C07272=1088.319,-113.427,-50.311,174.390,16.610,152.665
C07273=1088.312,-113.696,-50.301,174.388,16.610,152.665
C07274=1088.306,-113.946,-50.291,174.386,16.608,152.665
C07275=1088.300,-114.196,-50.282,174.384,16.608,152.666
C07276=1088.294,-114.446,-50.272,174.383,16.608,152.666
C07277=1088.288,-114.696,-50.263,174.381,16.607,152.666
C07278=1088.282,-114.945,-50.253,174.380,16.606,152.666
C07279=1088.275,-115.195,-50.244,174.378,16.605,152.666
C07280=1088.269,-115.445,-50.234,174.377,16.605,152.667
C07281=1088.263,-115.695,-50.224,174.375,16.604,152.667
C07282=1088.257,-115.945,-50.215,174.373,16.603,152.667
C07283=1088.251,-116.194,-50.205,174.372,16.603,152.667
C07284=1088.245,-116.444,-50.196,174.370,16.603,152.667
C07285=1088.239,-116.693,-50.187,174.369,16.602,152.668
C07286=1088.233,-116.943,-50.177,174.368,16.602,152.668
C07287=1088.227,-117.193,-50.167,174.366,16.601,152.668
C07288=1088.220,-117.443,-50.158,174.364,16.600,152.668
C07289=1088.215,-117.693,-50.149,174.363,16.600,152.668
C07290=1088.208,-117.943,-50.139,174.361,16.599,152.669
C07291=1088.202,-118.193,-50.130,174.359,16.598,152.669
C07292=1088.197,-118.442,-50.121,174.358,16.598,152.669
C07293=1088.190,-118.691,-50.112,174.356,16.597,152.669
C07294=1088.184,-118.941,-50.102,174.355,16.596,152.669
C07295=1088.177,-119.191,-50.093,174.354,16.596,152.670
C07296=1088.171,-119.441,-50.083,174.352,16.596,152.670
C07297=1088.165,-119.691,-50.073,174.350,16.595,152.670
C07298=1088.159,-119.941,-50.065,174.348,16.594,152.670
C07299=1088.153,-120.191,-50.055,174.347,16.594,152.670
C07300=1088.147,-120.440,-50.046,174.345,16.593,152.671
C07301=1088.141,-120.689,-50.037,174.343,16.592,152.671
C07302=1088.134,-120.939,-50.027,174.342,16.592,152.671
C07303=1088.128,-121.189,-50.018,174.340,16.592,152.671
C07304=1088.122,-121.439,-50.009,174.340,16.591,152.671
C07305=1088.116,-121.689,-49.999,174.338,16.590,152.672
C07306=1088.110,-121.939,-49.990,174.336,16.590,152.672
C07307=1088.104,-122.188,-49.981,174.335,16.590,152.672
C07308=1088.098,-122.438,-49.972,174.333,16.589,152.672
C07309=1088.091,-122.687,-49.962,174.331,16.588,152.673
C07310=1088.086,-122.938,-49.953,174.330,16.588,152.673
C07311=1088.079,-123.188,-49.944,174.328,16.587,152.673
C07312=1088.074,-123.437,-49.934,174.326,16.586,152.673
C07313=1088.068,-123.686,-49.925,174.325,16.586,152.673
C07314=1088.061,-123.937,-49.917,174.323,16.586,152.674
C07315=1088.055,-124.186,-49.907,174.322,16.585,152.674
C07316=1088.049,-124.436,-49.897,174.321,16.585,152.674
C07317=1088.042,-124.686,-49.888,174.319,16.584,152.674
C07318=1088.037,-124.936,-49.879,174.317,16.583,152.674
C07319=1088.030,-125.185,-49.870,174.316,16.583,152.675
C07320=1088.024,-125.435,-49.861,174.314,16.583,152.675
C07321=1088.018,-125.685,-49.851,174.312,16.582,152.675
C07322=1088.012,-125.935,-49.842,174.311,16.582,152.675
C07323=1088.006,-126.184,-49.834,174.309,16.581,152.676
C07324=1088.000,-126.434,-49.824,174.308,16.581,152.676
C07325=1087.993,-126.684,-49.815,174.306,16.580,152.676
C07326=1087.987,-126.934,-49.806,174.304,16.580,152.676
C07327=1087.981,-127.183,-49.797,174.303,16.580,152.677
C07328=1087.974,-127.433,-49.787,174.302,16.579,152.677
C07329=1087.969,-127.683,-49.779,174.300,16.578,152.677
C07330=1087.962,-127.941,-49.769,174.299,16.578,152.677
C07331=1087.957,-128.198,-49.760,174.297,16.577,152.677
C07332=1087.958,-128.455,-49.748,174.296,16.575,152.677
C07333=1087.965,-128.710,-49.735,174.296,16.571,152.676
C07334=1087.560,-128.731,-49.860,174.254,16.677,152.705
C07335=1087.553,-128.477,-49.873,174.254,16.681,152.706
C07336=1087.552,-128.220,-49.885,174.255,16.683,152.706
C07337=1087.558,-127.963,-49.895,174.257,16.684,152.706
C07338=1087.564,-127.705,-49.904,174.258,16.684,152.705
C07339=1087.571,-127.455,-49.914,174.260,16.685,152.705
C07340=1087.576,-127.205,-49.922,174.262,16.686,152.705
C07341=1087.582,-126.955,-49.932,174.263,16.686,152.705
C07342=1087.589,-126.706,-49.941,174.265,16.687,152.705
C07343=1087.595,-126.456,-49.950,174.267,16.687,152.704
C07344=1087.601,-126.206,-49.959,174.268,16.687,152.704
C07345=1087.607,-125.957,-49.969,174.270,16.688,152.704
C07346=1087.614,-125.707,-49.978,174.271,16.689,152.704
C07347=1087.619,-125.457,-49.986,174.272,16.689,152.703
C07348=1087.626,-125.207,-49.996,174.274,16.690,152.703
C07349=1087.632,-124.957,-50.005,174.275,16.690,152.703
C07350=1087.639,-124.708,-50.014,174.277,16.691,152.703
C07351=1087.644,-124.458,-50.023,174.279,16.691,152.703
C07352=1087.650,-124.208,-50.033,174.280,16.691,152.702
C07353=1087.656,-123.958,-50.042,174.282,16.692,152.702
C07354=1087.663,-123.709,-50.051,174.284,16.693,152.702
C07355=1087.669,-123.458,-50.060,174.285,16.693,152.702
C07356=1087.675,-123.209,-50.069,174.287,16.694,152.701
C07357=1087.681,-122.960,-50.079,174.289,16.694,152.701
C07358=1087.687,-122.710,-50.088,174.289,16.695,152.701
C07359=1087.693,-122.460,-50.098,174.291,16.696,152.701
C07360=1087.700,-122.210,-50.106,174.293,16.696,152.701
C07361=1087.706,-121.960,-50.116,174.294,16.697,152.701
C07362=1087.711,-121.711,-50.125,174.296,16.697,152.700
C07363=1087.718,-121.461,-50.134,174.298,16.698,152.700
C07364=1087.724,-121.211,-50.144,174.299,16.698,152.700
C07365=1087.730,-120.961,-50.153,174.301,16.699,152.700
C07366=1087.736,-120.711,-50.162,174.303,16.700,152.699
C07367=1087.743,-120.462,-50.171,174.304,16.700,152.699
C07368=1087.748,-120.213,-50.181,174.305,16.701,152.699
C07369=1087.754,-119.963,-50.190,174.307,16.701,152.699
C07370=1087.761,-119.713,-50.200,174.308,16.701,152.699
C07371=1087.767,-119.463,-50.209,174.310,16.702,152.698
C07372=1087.773,-119.213,-50.218,174.312,16.703,152.698
C07373=1087.779,-118.963,-50.228,174.313,16.703,152.698
C07374=1087.785,-118.713,-50.237,174.315,16.704,152.698
C07375=1087.792,-118.464,-50.246,174.316,16.705,152.698
C07376=1087.798,-118.215,-50.255,174.318,16.705,152.697
C07377=1087.804,-117.965,-50.265,174.319,16.706,152.697
C07378=1087.810,-117.715,-50.275,174.321,16.706,152.697
C07379=1087.816,-117.465,-50.284,174.323,16.708,152.697
C07380=1087.822,-117.215,-50.294,174.324,16.708,152.697
C07381=1087.828,-116.966,-50.303,174.326,16.708,152.696
C07382=1087.835,-116.716,-50.313,174.327,16.709,152.696
C07383=1087.840,-116.465,-50.322,174.329,16.709,152.696
C07384=1087.847,-116.216,-50.331,174.330,16.710,152.696
C07385=1087.852,-115.967,-50.340,174.332,16.711,152.696
C07386=1087.858,-115.717,-50.350,174.333,16.711,152.696
C07387=1087.864,-115.467,-50.360,174.335,16.712,152.695
C07388=1087.871,-115.217,-50.369,174.337,16.713,152.695
C07389=1087.877,-114.967,-50.379,174.338,16.714,152.695
C07390=1087.883,-114.718,-50.388,174.339,16.714,152.695
C07391=1087.889,-114.468,-50.398,174.341,16.714,152.695
C07392=1087.895,-114.218,-50.407,174.343,16.716,152.694
C07393=1087.902,-113.968,-50.417,174.344,16.716,152.694
C07394=1087.908,-113.718,-50.427,174.346,16.717,152.694
C07395=1087.915,-113.448,-50.437,174.348,16.717,152.694
C07396=1087.921,-113.177,-50.447,174.349,16.718,152.694
C07397=1087.928,-112.907,-50.458,174.351,16.719,152.693
C07398=1087.934,-112.635,-50.468,174.353,16.720,152.693
C07399=1087.940,-112.385,-50.477,174.354,16.720,152.693
C07400=1087.947,-112.135,-50.487,174.356,16.721,152.693
C07401=1087.953,-111.886,-50.497,174.358,16.722,152.693
C07402=1087.959,-111.636,-50.506,174.359,16.722,152.693
C07403=1087.964,-111.387,-50.515,174.360,16.723,152.692
C07404=1087.971,-111.137,-50.525,174.362,16.724,152.692
C07405=1087.977,-110.887,-50.534,174.364,16.725,152.692
C07406=1087.983,-110.638,-50.545,174.365,16.725,152.692
C07407=1087.989,-110.388,-50.554,174.367,16.726,152.692
C07408=1087.995,-110.138,-50.564,174.368,16.726,152.691
C07409=1088.001,-109.888,-50.574,174.369,16.727,152.691
C07410=1088.007,-109.639,-50.584,174.371,16.728,152.691
C07411=1088.013,-109.389,-50.593,174.373,16.729,152.691
C07412=1088.020,-109.139,-50.603,174.375,16.729,152.691
C07413=1088.026,-108.889,-50.612,174.376,16.730,152.691
C07414=1088.032,-108.639,-50.622,174.377,16.730,152.690
C07415=1088.038,-108.390,-50.631,174.379,16.731,152.690
C07416=1088.045,-108.140,-50.642,174.381,16.732,152.690
C07417=1088.051,-107.891,-50.651,174.382,16.733,152.690
C07418=1088.057,-107.641,-50.661,174.383,16.734,152.690
C07419=1088.062,-107.391,-50.671,174.385,16.734,152.690
C07420=1088.068,-107.141,-50.681,174.387,16.735,152.689
C07421=1088.075,-106.891,-50.690,174.388,16.735,152.689
C07422=1088.081,-106.642,-50.700,174.390,16.737,152.689
C07423=1088.087,-106.392,-50.710,174.392,16.737,152.689
C07424=1088.093,-106.142,-50.720,174.393,16.738,152.689
C07425=1088.099,-105.892,-50.730,174.394,16.739,152.689
C07426=1088.105,-105.642,-50.739,174.396,16.739,152.688
C07427=1088.111,-105.393,-50.749,174.398,16.740,152.688
C07428=1088.118,-105.143,-50.759,174.400,16.741,152.688
C07429=1088.123,-104.893,-50.769,174.400,16.742,152.688
C07430=1088.129,-104.643,-50.779,174.402,16.743,152.688
C07431=1088.136,-104.394,-50.788,174.404,16.743,152.688
C07432=1088.142,-104.145,-50.799,174.406,16.744,152.687
C07433=1088.147,-103.894,-50.809,174.407,16.746,152.687
C07434=1088.154,-103.645,-50.818,174.408,16.746,152.687
C07435=1088.160,-103.395,-50.828,174.410,16.747,152.687
C07436=1088.166,-103.145,-50.838,174.412,16.747,152.687
C07437=1088.172,-102.896,-50.848,174.413,16.748,152.687
C07438=1088.178,-102.646,-50.858,174.414,16.749,152.687
C07439=1088.184,-102.396,-50.868,174.416,16.750,152.686
C07440=1088.190,-102.147,-50.878,174.418,16.751,152.686
C07441=1088.196,-101.897,-50.888,174.419,16.752,152.686
C07442=1088.202,-101.647,-50.898,174.421,16.752,152.686
C07443=1088.208,-101.397,-50.907,174.422,16.753,152.686
C07444=1088.215,-101.148,-50.917,174.424,16.754,152.686
C07445=1088.220,-100.898,-50.928,174.426,16.755,152.685
C07446=1088.226,-100.648,-50.937,174.427,16.756,152.685
C07447=1088.233,-100.399,-50.947,174.428,16.756,152.685
C07448=1088.238,-100.149,-50.958,174.430,16.757,152.685
C07449=1088.244,-99.899,-50.967,174.432,16.758,152.685
C07450=1088.251,-99.650,-50.977,174.433,16.759,152.685
C07451=1088.257,-99.400,-50.987,174.435,16.760,152.684
C07452=1088.263,-99.150,-50.997,174.436,16.760,152.684
C07453=1088.269,-98.901,-51.008,174.438,16.761,152.684
C07454=1088.275,-98.651,-51.017,174.440,16.762,152.684
C07455=1088.281,-98.401,-51.027,174.441,16.763,152.684
C07456=1088.288,-98.151,-51.038,174.443,16.764,152.684
C07457=1088.294,-97.901,-51.047,174.444,16.765,152.684
C07458=1088.300,-97.652,-51.058,174.446,16.765,152.684
C07459=1088.306,-97.375,-51.069,174.447,16.766,152.683
C07460=1088.312,-97.099,-51.080,174.449,16.767,152.683
C07461=1088.319,-96.822,-51.091,174.451,16.769,152.683
C07462=1088.326,-96.546,-51.103,174.452,16.769,152.683
C07463=1088.331,-96.296,-51.113,174.454,16.770,152.683
C07464=1088.338,-96.047,-51.123,174.456,16.771,152.683
C07465=1088.343,-95.796,-51.133,174.457,16.772,152.683
C07466=1088.349,-95.547,-51.143,174.458,16.773,152.683
C07467=1088.356,-95.296,-51.154,174.460,16.774,152.682
C07468=1088.362,-95.047,-51.164,174.462,16.775,152.682
C07469=1088.368,-94.797,-51.174,174.463,16.776,152.682
C07470=1088.374,-94.547,-51.184,174.465,16.777,152.682
C07471=1088.380,-94.298,-51.194,174.467,16.778,152.682
C07472=1088.386,-94.048,-51.205,174.468,16.778,152.682
C07473=1088.392,-93.799,-51.215,174.469,16.779,152.681
C07474=1088.398,-93.549,-51.225,174.471,16.780,152.681
C07475=1088.403,-93.299,-51.235,174.473,16.781,152.681
C07476=1088.410,-93.050,-51.245,174.474,16.782,152.681
C07477=1088.415,-92.799,-51.256,174.476,16.784,152.681
C07478=1088.422,-92.550,-51.266,174.477,16.784,152.681
C07479=1088.427,-92.300,-51.276,174.479,16.785,152.681
C07480=1088.434,-92.050,-51.287,174.480,16.786,152.681
C07481=1088.440,-91.801,-51.298,174.482,16.787,152.680
C07482=1088.446,-91.551,-51.307,174.484,16.788,152.680
C07483=1088.452,-91.301,-51.318,174.485,16.789,152.680
C07484=1088.458,-91.052,-51.328,174.486,16.789,152.680
C07485=1088.464,-90.802,-51.338,174.488,16.790,152.680
C07486=1088.470,-90.552,-51.348,174.490,16.791,152.680
C07487=1088.475,-90.303,-51.359,174.491,16.792,152.680
C07488=1088.482,-90.053,-51.368,174.493,16.794,152.680
C07489=1088.488,-89.803,-51.380,174.494,16.795,152.679
C07490=1088.494,-89.553,-51.391,174.495,16.795,152.679
C07491=1088.500,-89.304,-51.400,174.497,16.796,152.679
C07492=1088.506,-89.054,-51.411,174.499,16.797,152.679
C07493=1088.512,-88.804,-51.421,174.500,16.798,152.679
C07494=1088.518,-88.555,-51.431,174.502,16.799,152.679
C07495=1088.524,-88.306,-51.442,174.504,16.800,152.679
C07496=1088.530,-88.055,-51.452,174.505,16.801,152.679
C07497=1088.537,-87.806,-51.463,174.506,16.802,152.679
C07498=1088.542,-87.556,-51.473,174.508,16.803,152.678
C07499=1088.548,-87.306,-51.484,174.509,16.804,152.678
C07500=1088.554,-87.057,-51.494,174.511,16.805,152.678
C07501=1088.560,-86.806,-51.504,174.513,16.806,152.678
C07502=1088.567,-86.557,-51.515,174.515,16.807,152.678
C07503=1088.572,-86.307,-51.526,174.516,16.808,152.678
C07504=1088.578,-86.057,-51.536,174.517,16.809,152.678
C07505=1088.584,-85.808,-51.546,174.519,16.810,152.678
C07506=1088.590,-85.559,-51.557,174.520,16.811,152.677
C07507=1088.597,-85.308,-51.567,174.522,16.812,152.677
C07508=1088.603,-85.059,-51.578,174.524,16.813,152.677
C07509=1088.608,-84.809,-51.589,174.525,16.814,152.677
C07510=1088.615,-84.560,-51.599,174.527,16.815,152.677
C07511=1088.621,-84.309,-51.609,174.529,16.816,152.677
C07512=1088.627,-84.060,-51.620,174.530,16.816,152.677
C07513=1088.633,-83.810,-51.631,174.531,16.817,152.677
C07514=1088.639,-83.560,-51.641,174.533,16.819,152.676
C07515=1088.645,-83.311,-51.651,174.534,16.820,152.676
C07516=1088.651,-83.061,-51.662,174.536,16.821,152.676
C07517=1088.657,-82.812,-51.673,174.538,16.822,152.676
C07518=1088.663,-82.562,-51.683,174.539,16.823,152.676
C07519=1088.669,-82.312,-51.694,174.541,16.824,152.676
C07520=1088.676,-82.062,-51.704,174.542,16.825,152.676
C07521=1088.682,-81.813,-51.715,174.543,16.826,152.676
C07522=1088.688,-81.563,-51.726,174.545,16.827,152.676
C07523=1088.695,-81.289,-51.737,174.547,16.828,152.676
C07524=1088.701,-81.015,-51.749,174.548,16.829,152.675
C07525=1088.707,-80.740,-51.761,174.551,16.831,152.675
C07526=1088.715,-80.466,-51.772,174.553,16.831,152.675
C07527=1088.721,-80.216,-51.783,174.553,16.832,152.675
C07528=1088.727,-79.966,-51.793,174.555,16.833,152.675
C07529=1088.733,-79.717,-51.804,174.557,16.834,152.675
C07530=1088.739,-79.467,-51.815,174.558,16.835,152.675
C07531=1088.745,-79.217,-51.826,174.560,16.836,152.675
C07532=1088.751,-78.968,-51.837,174.561,16.838,152.675
C07533=1088.756,-78.718,-51.848,174.563,16.839,152.674
C07534=1088.763,-78.468,-51.857,174.565,16.840,152.674
C07535=1088.769,-78.218,-51.869,174.566,16.841,152.674
C07536=1088.775,-77.969,-51.879,174.568,16.842,152.674
C07537=1088.780,-77.719,-51.890,174.570,16.843,152.674
C07538=1088.786,-77.470,-51.901,174.570,16.844,152.674
C07539=1088.793,-77.220,-51.912,174.572,16.845,152.674
C07540=1088.799,-76.970,-51.923,174.574,16.846,152.674
C07541=1088.805,-76.721,-51.934,174.575,16.847,152.674
C07542=1088.810,-76.471,-51.945,174.577,16.848,152.674
C07543=1088.816,-76.220,-51.955,174.578,16.850,152.673
C07544=1088.822,-75.971,-51.966,174.580,16.851,152.673
C07545=1088.828,-75.722,-51.977,174.582,16.852,152.673
C07546=1088.835,-75.472,-51.987,174.583,16.853,152.673
C07547=1088.841,-75.222,-51.998,174.585,16.854,152.673
C07548=1088.846,-74.973,-52.009,174.587,16.855,152.673
C07549=1088.852,-74.723,-52.020,174.588,16.856,152.673
C07550=1088.859,-74.473,-52.031,174.590,16.858,152.673
C07551=1088.864,-74.223,-52.042,174.591,16.859,152.673
C07552=1088.870,-73.974,-52.053,174.592,16.859,152.673
C07553=1088.876,-73.724,-52.064,174.594,16.861,152.673
C07554=1088.882,-73.474,-52.075,174.595,16.862,152.672
C07555=1088.888,-73.225,-52.086,174.597,16.863,152.672
C07556=1088.894,-72.975,-52.097,174.599,16.864,152.672
C07557=1088.900,-72.725,-52.108,174.600,16.865,152.672
C07558=1088.906,-72.476,-52.119,174.602,16.867,152.672
C07559=1088.911,-72.226,-52.130,174.603,16.868,152.672
C07560=1088.917,-71.977,-52.141,174.605,16.869,152.672
C07561=1088.923,-71.726,-52.152,174.606,16.870,152.672
C07562=1088.929,-71.477,-52.163,174.608,16.871,152.672
C07563=1088.935,-71.228,-52.174,174.609,16.873,152.672
C07564=1088.941,-70.978,-52.185,174.611,16.874,152.672
C07565=1088.947,-70.728,-52.196,174.613,16.875,152.672
C07566=1088.953,-70.478,-52.207,174.614,16.876,152.671
C07567=1088.958,-70.229,-52.218,174.616,16.877,152.671
C07568=1088.964,-69.978,-52.230,174.617,16.879,152.671
C07569=1088.970,-69.729,-52.240,174.619,16.880,152.671
C07570=1088.976,-69.479,-52.251,174.621,16.881,152.671
C07571=1088.982,-69.230,-52.263,174.622,16.882,152.671
C07572=1088.988,-68.980,-52.274,174.623,16.883,152.671
C07573=1088.994,-68.731,-52.285,174.624,16.884,152.671
C07574=1088.999,-68.481,-52.296,174.626,16.885,152.671
C07575=1089.006,-68.231,-52.307,174.628,16.886,152.671
C07576=1089.012,-67.982,-52.318,174.629,16.887,152.671
C07577=1089.017,-67.732,-52.329,174.631,16.889,152.671
C07578=1089.023,-67.482,-52.341,174.632,16.890,152.671
C07579=1089.029,-67.232,-52.352,174.634,16.891,152.671
C07580=1089.035,-66.983,-52.364,174.636,16.892,152.670
C07581=1089.041,-66.733,-52.374,174.637,16.893,152.670
C07582=1089.047,-66.484,-52.385,174.639,16.895,152.670
C07583=1089.053,-66.233,-52.397,174.640,16.896,152.670
C07584=1089.059,-65.984,-52.407,174.642,16.897,152.670
C07585=1089.065,-65.734,-52.418,174.643,16.898,152.670
C07586=1089.071,-65.485,-52.430,174.645,16.900,152.670
C07587=1089.077,-65.213,-52.443,174.646,16.901,152.670
C07588=1089.084,-64.941,-52.455,174.648,16.902,152.670
C07589=1089.090,-64.668,-52.467,174.650,16.904,152.670
C07590=1089.097,-64.396,-52.479,174.652,16.905,152.670
C07591=1089.102,-64.147,-52.490,174.654,16.906,152.669
C07592=1089.109,-63.897,-52.501,174.655,16.908,152.670
C07593=1089.114,-63.647,-52.513,174.657,16.909,152.669
C07594=1089.120,-63.398,-52.525,174.658,16.910,152.669
C07595=1089.126,-63.148,-52.536,174.660,16.911,152.669
C07596=1089.132,-62.898,-52.547,174.661,16.913,152.669
C07597=1089.138,-62.648,-52.558,174.663,16.914,152.669
C07598=1089.144,-62.399,-52.570,174.665,16.915,152.669
C07599=1089.150,-62.149,-52.581,174.666,16.916,152.669
C07600=1089.156,-61.899,-52.592,174.668,16.918,152.669
C07601=1089.162,-61.650,-52.604,174.669,16.919,152.669
C07602=1089.168,-61.400,-52.615,174.671,16.920,152.669
C07603=1089.174,-61.151,-52.626,174.672,16.921,152.669
C07604=1089.180,-60.901,-52.638,174.674,16.922,152.669
C07605=1089.185,-60.651,-52.649,174.675,16.924,152.669
C07606=1089.192,-60.401,-52.661,174.677,16.925,152.668
C07607=1089.198,-60.152,-52.672,174.679,16.926,152.668
C07608=1089.204,-59.902,-52.683,174.680,16.927,152.668
C07609=1089.210,-59.653,-52.694,174.682,16.929,152.668
C07610=1089.215,-59.403,-52.707,174.683,16.930,152.668
C07611=1089.222,-59.153,-52.718,174.685,16.931,152.668
C07612=1089.227,-58.904,-52.729,174.686,16.932,152.668
C07613=1089.234,-58.654,-52.741,174.688,16.933,152.668
C07614=1089.239,-58.404,-52.752,174.690,16.935,152.668
C07615=1089.245,-58.154,-52.763,174.691,16.936,152.668
C07616=1089.251,-57.905,-52.775,174.693,16.937,152.668
C07617=1089.258,-57.655,-52.786,174.694,16.938,152.668
C07618=1089.264,-57.406,-52.798,174.696,16.939,152.668
C07619=1089.269,-57.156,-52.810,174.697,16.941,152.668
C07620=1089.275,-56.907,-52.821,174.699,16.942,152.668
C07621=1089.282,-56.657,-52.832,174.700,16.943,152.667
C07622=1089.287,-56.407,-52.843,174.702,16.944,152.667
C07623=1089.293,-56.157,-52.856,174.704,16.946,152.667
C07624=1089.300,-55.907,-52.867,174.705,16.947,152.667
C07625=1089.306,-55.658,-52.879,174.707,16.948,152.667
C07626=1089.312,-55.408,-52.890,174.708,16.949,152.667
C07627=1089.317,-55.159,-52.902,174.710,16.951,152.667
C07628=1089.324,-54.909,-52.913,174.711,16.952,152.667
C07629=1089.330,-54.660,-52.925,174.713,16.953,152.667
C07630=1089.336,-54.410,-52.936,174.715,16.954,152.667
C07631=1089.341,-54.161,-52.948,174.716,16.956,152.667
C07632=1089.348,-53.910,-52.960,174.718,16.957,152.667
C07633=1089.354,-53.661,-52.972,174.719,16.958,152.667
C07634=1089.360,-53.411,-52.982,174.721,16.959,152.667
C07635=1089.366,-53.161,-52.995,174.722,16.961,152.667
C07636=1089.372,-52.912,-53.006,174.724,16.962,152.666
C07637=1089.378,-52.662,-53.018,174.725,16.963,152.666
C07638=1089.383,-52.412,-53.029,174.727,16.965,152.666
C07639=1089.390,-52.163,-53.041,174.728,16.966,152.666
C07640=1089.396,-51.913,-53.053,174.730,16.967,152.666
C07641=1089.402,-51.664,-53.065,174.732,16.968,152.666
C07642=1089.408,-51.414,-53.077,174.734,16.970,152.666
C07643=1089.414,-51.164,-53.088,174.735,16.971,152.666
C07644=1089.421,-50.915,-53.100,174.737,16.972,152.666
C07645=1089.426,-50.664,-53.111,174.738,16.974,152.666
C07646=1089.432,-50.416,-53.123,174.740,16.975,152.666
C07647=1089.438,-50.166,-53.135,174.742,16.976,152.666
C07648=1089.444,-49.916,-53.146,174.743,16.978,152.666
C07649=1089.450,-49.666,-53.159,174.745,16.979,152.666
C07650=1089.456,-49.417,-53.170,174.746,16.980,152.666
C07651=1089.462,-49.146,-53.184,174.748,16.982,152.666
C07652=1089.469,-48.875,-53.196,174.749,16.983,152.666
C07653=1089.474,-48.604,-53.209,174.751,16.985,152.666
C07654=1089.481,-48.334,-53.221,174.753,16.986,152.665
C07655=1089.487,-48.084,-53.234,174.754,16.988,152.665
C07656=1089.494,-47.834,-53.246,174.756,16.989,152.665
C07657=1089.499,-47.584,-53.257,174.758,16.990,152.665
C07658=1089.505,-47.335,-53.269,174.759,16.991,152.665
C07659=1089.510,-47.086,-53.282,174.761,16.992,152.665
C07660=1089.517,-46.835,-53.293,174.762,16.994,152.665
C07661=1089.522,-46.586,-53.305,174.764,16.995,152.665
C07662=1089.529,-46.337,-53.317,174.765,16.996,152.665
C07663=1089.534,-46.086,-53.329,174.768,16.998,152.665
C07664=1089.540,-45.837,-53.341,174.769,17.000,152.665
C07665=1089.546,-45.587,-53.353,174.770,17.001,152.665
C07666=1089.552,-45.338,-53.365,174.772,17.002,152.665
C07667=1089.558,-45.088,-53.376,174.774,17.003,152.665
C07668=1089.564,-44.838,-53.389,174.775,17.005,152.665
C07669=1089.569,-44.589,-53.401,174.777,17.006,152.665
C07670=1089.576,-44.339,-53.413,174.778,17.008,152.665
C07671=1089.581,-44.089,-53.425,174.780,17.009,152.665
C07672=1089.587,-43.840,-53.436,174.781,17.010,152.665
C07673=1089.593,-43.590,-53.449,174.783,17.012,152.665
C07674=1089.599,-43.341,-53.461,174.784,17.013,152.664
C07675=1089.605,-43.091,-53.473,174.786,17.014,152.665
C07676=1089.611,-42.841,-53.485,174.788,17.016,152.664
C07677=1089.617,-42.592,-53.497,174.789,17.018,152.664
C07678=1089.623,-42.342,-53.509,174.791,17.019,152.664
C07679=1089.629,-42.092,-53.522,174.793,17.020,152.664
C07680=1089.635,-41.843,-53.533,174.794,17.021,152.664
C07681=1089.640,-41.593,-53.545,174.796,17.022,152.664
C07682=1089.646,-41.343,-53.558,174.797,17.024,152.664
C07683=1089.652,-41.094,-53.569,174.799,17.025,152.664
C07684=1089.658,-40.844,-53.582,174.800,17.026,152.664
C07685=1089.665,-40.595,-53.594,174.802,17.028,152.664
C07686=1089.670,-40.345,-53.606,174.803,17.029,152.664
C07687=1089.676,-40.096,-53.619,174.806,17.031,152.664
C07688=1089.683,-39.845,-53.630,174.807,17.032,152.664
C07689=1089.688,-39.596,-53.642,174.809,17.034,152.664
C07690=1089.694,-39.346,-53.655,174.810,17.035,152.664
C07691=1089.700,-39.097,-53.666,174.812,17.036,152.664
C07692=1089.706,-38.847,-53.679,174.813,17.038,152.664
C07693=1089.712,-38.598,-53.691,174.815,17.039,152.664
C07694=1089.717,-38.348,-53.704,174.816,17.040,152.664
C07695=1089.724,-38.098,-53.716,174.818,17.042,152.664
C07696=1089.729,-37.849,-53.728,174.820,17.044,152.664
C07697=1089.735,-37.599,-53.740,174.822,17.045,152.663
C07698=1089.741,-37.349,-53.753,174.823,17.046,152.663
C07699=1089.747,-37.100,-53.765,174.825,17.048,152.663
C07700=1089.753,-36.851,-53.777,174.826,17.049,152.663
C07701=1089.759,-36.601,-53.790,174.828,17.050,152.663
C07702=1089.764,-36.351,-53.802,174.829,17.052,152.663
C07703=1089.770,-36.102,-53.814,174.831,17.053,152.663
C07704=1089.776,-35.852,-53.827,174.832,17.055,152.663
C07705=1089.781,-35.602,-53.838,174.834,17.056,152.663
C07706=1089.788,-35.352,-53.850,174.836,17.058,152.663
C07707=1089.794,-35.103,-53.864,174.837,17.059,152.663
C07708=1089.800,-34.853,-53.876,174.839,17.061,152.663
C07709=1089.805,-34.604,-53.888,174.840,17.062,152.663
C07710=1089.811,-34.354,-53.901,174.842,17.063,152.663
C07711=1089.817,-34.104,-53.914,174.843,17.064,152.663
C07712=1089.823,-33.854,-53.926,174.845,17.066,152.663
C07713=1089.829,-33.606,-53.938,174.847,17.068,152.663
C07714=1089.835,-33.356,-53.950,174.848,17.069,152.663
C07715=1089.841,-33.085,-53.964,174.850,17.070,152.663
C07716=1089.847,-32.815,-53.978,174.851,17.072,152.663
C07717=1089.854,-32.544,-53.991,174.854,17.074,152.663
C07718=1089.860,-32.273,-54.004,174.855,17.075,152.663
C07719=1089.866,-32.024,-54.017,174.857,17.076,152.663
C07720=1089.872,-31.774,-54.030,174.858,17.078,152.663
C07721=1089.878,-31.525,-54.042,174.860,17.079,152.663
C07722=1089.883,-31.275,-54.054,174.862,17.081,152.663
C07723=1089.889,-31.025,-54.067,174.864,17.082,152.663
C07724=1089.895,-30.775,-54.080,174.865,17.084,152.663
C07725=1089.901,-30.527,-54.091,174.867,17.085,152.662
C07726=1089.907,-30.277,-54.104,174.868,17.087,152.663
C07727=1089.913,-30.027,-54.117,174.870,17.088,152.662
C07728=1089.919,-29.778,-54.129,174.871,17.089,152.662
C07729=1089.925,-29.528,-54.142,174.873,17.091,152.662
C07730=1089.931,-29.278,-54.154,174.875,17.092,152.662
C07731=1089.937,-29.029,-54.167,174.876,17.094,152.662
C07732=1089.943,-28.779,-54.180,174.878,17.095,152.662
C07733=1089.949,-28.529,-54.193,174.879,17.096,152.662
C07734=1089.955,-28.280,-54.205,174.881,17.098,152.662
C07735=1089.960,-28.030,-54.218,174.882,17.099,152.662
C07736=1089.966,-27.780,-54.230,174.885,17.101,152.662
C07737=1089.972,-27.531,-54.243,174.886,17.102,152.662
C07738=1089.979,-27.282,-54.255,174.888,17.103,152.662
C07739=1089.985,-27.032,-54.268,174.889,17.105,152.662
C07740=1089.990,-26.782,-54.280,174.891,17.106,152.662
C07741=1089.996,-26.532,-54.294,174.892,17.108,152.662
C07742=1090.001,-26.283,-54.306,174.894,17.109,152.662
C07743=1090.007,-26.033,-54.319,174.896,17.111,152.662
C07744=1090.013,-25.783,-54.331,174.898,17.112,152.662
C07745=1090.019,-25.534,-54.345,174.899,17.114,152.662
C07746=1090.025,-25.284,-54.357,174.900,17.115,152.662
C07747=1090.030,-25.035,-54.369,174.902,17.116,152.662
C07748=1090.037,-24.786,-54.383,174.903,17.118,152.662
C07749=1090.043,-24.536,-54.395,174.906,17.120,152.662
C07750=1090.048,-24.286,-54.408,174.907,17.121,152.662
C07751=1090.054,-24.036,-54.421,174.909,17.122,152.662
C07752=1090.060,-23.787,-54.434,174.910,17.124,152.662
C07753=1090.065,-23.537,-54.446,174.912,17.125,152.662
C07754=1090.071,-23.287,-54.459,174.914,17.127,152.662
C07755=1090.077,-23.038,-54.472,174.915,17.129,152.662
C07756=1090.083,-22.788,-54.485,174.917,17.130,152.661
C07757=1090.089,-22.539,-54.498,174.918,17.132,152.662
C07758=1090.095,-22.289,-54.511,174.920,17.133,152.661
C07759=1090.100,-22.039,-54.524,174.921,17.134,152.661
C07760=1090.106,-21.790,-54.537,174.924,17.136,152.661
C07761=1090.112,-21.541,-54.549,174.925,17.138,152.661
C07762=1090.118,-21.291,-54.562,174.927,17.139,152.661
C07763=1090.124,-21.041,-54.575,174.928,17.140,152.661
C07764=1090.129,-20.791,-54.588,174.930,17.141,152.661
C07765=1090.136,-20.542,-54.601,174.931,17.143,152.661
C07766=1090.141,-20.292,-54.614,174.933,17.145,152.661
C07767=1090.148,-20.043,-54.627,174.935,17.146,152.661
C07768=1090.154,-19.793,-54.640,174.936,17.147,152.661
C07769=1090.158,-19.544,-54.653,174.938,17.149,152.661
C07770=1090.164,-19.294,-54.666,174.939,17.151,152.661
C07771=1090.170,-19.044,-54.678,174.942,17.152,152.661
C07772=1090.176,-18.795,-54.692,174.943,17.154,152.661
C07773=1090.182,-18.545,-54.704,174.945,17.155,152.661
C07774=1090.189,-18.296,-54.718,174.946,17.157,152.661
C07775=1090.194,-18.046,-54.731,174.948,17.158,152.661
C07776=1090.200,-17.796,-54.744,174.950,17.160,152.661
C07777=1090.206,-17.546,-54.756,174.951,17.161,152.661
C07778=1090.212,-17.297,-54.770,174.953,17.163,152.661
C07779=1090.218,-17.026,-54.784,174.954,17.164,152.661
C07780=1090.225,-16.755,-54.798,174.957,17.166,152.661
C07781=1090.231,-16.484,-54.812,174.958,17.167,152.661
C07782=1090.237,-16.213,-54.827,174.960,17.169,152.661
C07783=1090.243,-15.963,-54.840,174.962,17.170,152.661
C07784=1090.249,-15.713,-54.853,174.963,17.172,152.661
C07785=1090.255,-15.464,-54.865,174.965,17.173,152.661
C07786=1090.261,-15.214,-54.879,174.966,17.175,152.661
C07787=1090.267,-14.964,-54.892,174.968,17.176,152.661
C07788=1090.273,-14.715,-54.905,174.970,17.178,152.660
C07789=1090.278,-14.465,-54.919,174.972,17.179,152.661
C07790=1090.284,-14.215,-54.931,174.973,17.181,152.660
C07791=1090.290,-13.966,-54.945,174.975,17.182,152.660
C07792=1090.296,-13.716,-54.959,174.977,17.184,152.660
C07793=1090.302,-13.467,-54.971,174.978,17.185,152.660
C07794=1090.307,-13.217,-54.985,174.980,17.187,152.660
C07795=1090.313,-12.967,-54.998,174.981,17.188,152.660
C07796=1090.319,-12.718,-55.011,174.983,17.190,152.660
C07797=1090.325,-12.468,-55.025,174.985,17.191,152.660
C07798=1090.331,-12.218,-55.037,174.986,17.193,152.660
C07799=1090.336,-11.969,-55.051,174.988,17.194,152.660
C07800=1090.342,-11.720,-55.064,174.989,17.196,152.660
C07801=1090.348,-11.469,-55.078,174.991,17.197,152.660
C07802=1090.354,-11.220,-55.091,174.993,17.199,152.660
C07803=1090.359,-10.971,-55.105,174.995,17.201,152.660
C07804=1090.365,-10.721,-55.118,174.996,17.202,152.660
C07805=1090.371,-10.471,-55.130,174.998,17.203,152.660
C07806=1090.377,-10.222,-55.144,175.000,17.205,152.660
C07807=1090.383,-9.973,-55.158,175.001,17.207,152.660
C07808=1090.388,-9.722,-55.171,175.003,17.208,152.660
C07809=1090.394,-9.473,-55.184,175.004,17.209,152.660
C07810=1090.400,-9.224,-55.198,175.006,17.211,152.660
C07811=1090.406,-8.974,-55.211,175.008,17.212,152.660
C07812=1090.411,-8.724,-55.224,175.010,17.214,152.660
C07813=1090.418,-8.475,-55.238,175.011,17.215,152.660
C07814=1090.423,-8.225,-55.251,175.013,17.217,152.660
C07815=1090.429,-7.976,-55.265,175.015,17.218,152.660
C07816=1090.435,-7.727,-55.278,175.016,17.220,152.660
C07817=1090.441,-7.477,-55.291,175.018,17.221,152.660
C07818=1090.447,-7.227,-55.304,175.019,17.223,152.660
C07819=1090.452,-6.978,-55.318,175.022,17.224,152.660
C07820=1090.459,-6.728,-55.332,175.023,17.226,152.660
C07821=1090.464,-6.479,-55.345,175.025,17.228,152.660
C07822=1090.470,-6.230,-55.359,175.026,17.229,152.660
C07823=1090.476,-5.979,-55.372,175.028,17.230,152.660
C07824=1090.482,-5.729,-55.385,175.030,17.232,152.659
C07825=1090.488,-5.480,-55.399,175.031,17.234,152.660
C07826=1090.494,-5.231,-55.413,175.033,17.235,152.659
C07827=1090.499,-4.981,-55.426,175.034,17.236,152.660
C07828=1090.506,-4.732,-55.440,175.037,17.238,152.659
C07829=1090.511,-4.482,-55.454,175.038,17.240,152.659
C07830=1090.517,-4.233,-55.467,175.040,17.241,152.659
C07831=1090.523,-3.983,-55.481,175.041,17.242,152.659
C07832=1090.529,-3.733,-55.494,175.044,17.244,152.659
C07833=1090.535,-3.483,-55.508,175.045,17.246,152.659
C07834=1090.540,-3.234,-55.521,175.047,17.247,152.659
C07835=1090.546,-2.984,-55.535,175.048,17.248,152.659
C07836=1090.552,-2.735,-55.549,175.050,17.250,152.659
C07837=1090.557,-2.485,-55.562,175.052,17.251,152.659
C07838=1090.563,-2.236,-55.576,175.053,17.253,152.659
C07839=1090.569,-1.986,-55.590,175.055,17.254,152.659
C07840=1090.575,-1.737,-55.603,175.057,17.256,152.659
C07841=1090.580,-1.487,-55.617,175.059,17.257,152.659
C07842=1090.586,-1.238,-55.631,175.060,17.259,152.659
C07843=1090.592,-0.964,-55.646,175.062,17.261,152.659
C07844=1090.599,-0.692,-55.661,175.064,17.262,152.659
C07845=1090.605,-0.418,-55.676,175.066,17.264,152.659
C07846=1090.611,-0.146,-55.691,175.067,17.266,152.659
C07847=1090.617,0.103,-55.705,175.069,17.267,152.659
C07848=1090.623,0.353,-55.719,175.071,17.269,152.659
C07849=1090.628,0.603,-55.733,175.073,17.270,152.659
C07850=1090.635,0.852,-55.746,175.074,17.272,152.659
C07851=1090.640,1.102,-55.760,175.076,17.273,152.659
C07852=1090.645,1.351,-55.774,175.078,17.275,152.659
C07853=1090.651,1.601,-55.788,175.079,17.277,152.659
C07854=1090.656,1.851,-55.802,175.081,17.278,152.659
C07855=1090.663,2.100,-55.815,175.082,17.280,152.659
C07856=1090.669,2.350,-55.829,175.085,17.281,152.659
C07857=1090.674,2.600,-55.843,175.086,17.283,152.659
C07858=1090.680,2.849,-55.857,175.088,17.284,152.659
C07859=1090.685,3.098,-55.871,175.090,17.286,152.659
C07860=1090.692,3.347,-55.885,175.092,17.287,152.658
C07861=1090.697,3.597,-55.898,175.093,17.289,152.659
C07862=1090.703,3.847,-55.913,175.094,17.290,152.659
C07863=1090.709,4.097,-55.927,175.097,17.292,152.658
C07864=1090.714,4.346,-55.940,175.098,17.294,152.658
C07865=1090.721,4.595,-55.954,175.100,17.295,152.658
C07866=1090.726,4.845,-55.968,175.101,17.296,152.658
C07867=1090.732,5.094,-55.982,175.104,17.298,152.658
C07868=1090.738,5.345,-55.996,175.105,17.300,152.658
C07869=1090.743,5.594,-56.010,175.107,17.301,152.658
C07870=1090.749,5.844,-56.024,175.109,17.303,152.658
C07871=1090.755,6.092,-56.038,175.110,17.304,152.658
C07872=1090.761,6.343,-56.052,175.112,17.306,152.658
C07873=1090.767,6.592,-56.066,175.113,17.307,152.658
C07874=1090.772,6.842,-56.080,175.116,17.309,152.658
C07875=1090.778,7.091,-56.095,175.117,17.310,152.658
C07876=1090.783,7.340,-56.108,175.119,17.312,152.658
C07877=1090.790,7.590,-56.122,175.121,17.313,152.658
C07878=1090.796,7.840,-56.136,175.122,17.315,152.658
C07879=1090.802,8.089,-56.151,175.124,17.316,152.658
C07880=1090.807,8.338,-56.164,175.125,17.318,152.658
C07881=1090.813,8.589,-56.179,175.128,17.319,152.658
C07882=1090.819,8.838,-56.193,175.129,17.321,152.658
C07883=1090.824,9.087,-56.207,175.131,17.322,152.658
C07884=1090.830,9.337,-56.221,175.133,17.324,152.658
C07885=1090.837,9.587,-56.235,175.135,17.325,152.658
C07886=1090.842,9.836,-56.249,175.136,17.327,152.658
C07887=1090.848,10.085,-56.263,175.138,17.328,152.658
C07888=1090.854,10.335,-56.278,175.140,17.330,152.658
C07889=1090.860,10.584,-56.292,175.141,17.331,152.658
C07890=1090.865,10.834,-56.306,175.143,17.333,152.658
C07891=1090.872,11.084,-56.321,175.145,17.334,152.657
C07892=1090.877,11.333,-56.335,175.147,17.336,152.657
C07893=1090.883,11.583,-56.348,175.148,17.337,152.657
C07894=1090.889,11.833,-56.363,175.150,17.339,152.657
C07895=1090.894,12.082,-56.377,175.152,17.340,152.657
C07896=1090.901,12.331,-56.391,175.154,17.341,152.657
C07897=1090.907,12.581,-56.405,175.155,17.343,152.657
C07898=1090.913,12.831,-56.419,175.157,17.345,152.657
C07899=1090.918,13.080,-56.434,175.159,17.346,152.657
C07900=1090.924,13.330,-56.448,175.160,17.347,152.657
C07901=1090.930,13.579,-56.463,175.163,17.350,152.657
C07902=1090.936,13.828,-56.477,175.164,17.351,152.657
C07903=1090.942,14.078,-56.492,175.166,17.352,152.657
C07904=1090.947,14.328,-56.505,175.167,17.353,152.657
C07905=1090.953,14.577,-56.520,175.170,17.355,152.657
C07906=1090.959,14.827,-56.534,175.171,17.357,152.657
C07907=1090.965,15.102,-56.550,175.174,17.358,152.657
C07908=1090.972,15.376,-56.566,175.175,17.360,152.657
C07909=1090.977,15.651,-56.581,175.177,17.362,152.657
C07910=1090.985,15.926,-56.597,175.179,17.363,152.657
C07911=1090.991,16.175,-56.612,175.181,17.365,152.657
C07912=1090.995,16.425,-56.626,175.183,17.366,152.657
C07913=1091.002,16.675,-56.641,175.184,17.367,152.656
C07914=1091.007,16.924,-56.655,175.186,17.370,152.656
C07915=1091.013,17.173,-56.670,175.188,17.371,152.656
C07916=1091.019,17.423,-56.685,175.189,17.372,152.656
C07917=1091.025,17.673,-56.699,175.192,17.374,152.656
C07918=1091.031,17.922,-56.713,175.193,17.376,152.656
C07919=1091.037,18.172,-56.727,175.195,17.377,152.656
C07920=1091.042,18.421,-56.743,175.197,17.379,152.656
C07921=1091.048,18.671,-56.757,175.199,17.380,152.656
C07922=1091.054,18.920,-56.771,175.200,17.382,152.656
C07923=1091.059,19.169,-56.786,175.202,17.383,152.656
C07924=1091.065,19.420,-56.800,175.204,17.384,152.656
C07925=1091.071,19.669,-56.815,175.205,17.386,152.656
C07926=1091.076,19.918,-56.830,175.207,17.387,152.656
C07927=1091.082,20.168,-56.844,175.209,17.389,152.656
C07928=1091.088,20.417,-56.859,175.211,17.390,152.656
C07929=1091.094,20.667,-56.874,175.212,17.392,152.656
C07930=1091.100,20.916,-56.888,175.215,17.393,152.656
C07931=1091.105,21.166,-56.903,175.216,17.395,152.656
C07932=1091.111,21.415,-56.918,175.218,17.396,152.656
C07933=1091.117,21.665,-56.932,175.220,17.398,152.656
C07934=1091.123,21.914,-56.946,175.222,17.399,152.656
C07935=1091.128,22.164,-56.962,175.223,17.401,152.656
C07936=1091.134,22.413,-56.976,175.225,17.403,152.656
C07937=1091.140,22.663,-56.990,175.227,17.404,152.655
C07938=1091.145,22.912,-57.006,175.228,17.405,152.656
C07939=1091.152,23.162,-57.021,175.231,17.407,152.655
C07940=1091.157,23.411,-57.034,175.232,17.409,152.655
C07941=1091.163,23.661,-57.049,175.235,17.410,152.655
C07942=1091.168,23.910,-57.065,175.236,17.411,152.655
C07943=1091.174,24.159,-57.079,175.238,17.413,152.655
C07944=1091.180,24.410,-57.093,175.240,17.415,152.655
C07945=1091.185,24.659,-57.109,175.241,17.416,152.655
C07946=1091.192,24.909,-57.123,175.243,17.417,152.655
C07947=1091.197,25.158,-57.138,175.246,17.419,152.655
C07948=1091.203,25.407,-57.154,175.247,17.421,152.655
C07949=1091.209,25.657,-57.167,175.249,17.422,152.655
C07950=1091.215,25.907,-57.182,175.251,17.424,152.655
C07951=1091.220,26.156,-57.198,175.252,17.425,152.655
C07952=1091.226,26.406,-57.213,175.254,17.426,152.655
C07953=1091.232,26.655,-57.227,175.256,17.428,152.655
C07954=1091.238,26.905,-57.243,175.258,17.429,152.655
C07955=1091.243,27.154,-57.257,175.259,17.430,152.654
C07956=1091.250,27.404,-57.271,175.262,17.433,152.655
C07957=1091.255,27.653,-57.287,175.263,17.434,152.654
C07958=1091.261,27.903,-57.302,175.265,17.435,152.654
C07959=1091.267,28.152,-57.316,175.267,17.437,152.654
C07960=1091.273,28.402,-57.332,175.269,17.438,152.654
C07961=1091.278,28.651,-57.346,175.271,17.440,152.654
C07962=1091.284,28.901,-57.362,175.273,17.441,152.654
C07963=1091.290,29.150,-57.376,175.274,17.442,152.654
C07964=1091.295,29.399,-57.392,175.276,17.445,152.654
C07965=1091.301,29.648,-57.407,175.278,17.446,152.654
C07966=1091.306,29.898,-57.422,175.279,17.447,152.654
C07967=1091.312,30.148,-57.436,175.282,17.449,152.654
C07968=1091.317,30.397,-57.451,175.284,17.450,152.654
C07969=1091.324,30.647,-57.466,175.285,17.452,152.654
C07970=1091.329,30.896,-57.481,175.287,17.453,152.654
C07971=1091.336,31.172,-57.498,175.289,17.455,152.654
C07972=1091.342,31.449,-57.515,175.291,17.456,152.654
C07973=1091.348,31.725,-57.531,175.294,17.458,152.653
C07974=1091.354,32.002,-57.548,175.295,17.460,152.654
C07975=1091.361,32.250,-57.564,175.297,17.461,152.653
C07976=1091.366,32.500,-57.579,175.299,17.462,152.653
C07977=1091.372,32.749,-57.594,175.300,17.464,152.653
C07978=1091.378,32.999,-57.609,175.303,17.466,152.653
C07979=1091.384,33.249,-57.624,175.305,17.467,152.653
C07980=1091.389,33.498,-57.639,175.307,17.469,152.653
C07981=1091.395,33.748,-57.654,175.308,17.470,152.653
C07982=1091.401,33.997,-57.669,175.310,17.471,152.653
C07983=1091.407,34.247,-57.684,175.312,17.473,152.653
C07984=1091.412,34.496,-57.700,175.314,17.474,152.653
C07985=1091.418,34.746,-57.715,175.315,17.476,152.653
C07986=1091.424,34.996,-57.730,175.318,17.478,152.653
C07987=1091.429,35.245,-57.745,175.319,17.479,152.653
C07988=1091.436,35.494,-57.761,175.322,17.480,152.653
C07989=1091.441,35.743,-57.776,175.323,17.482,152.653
C07990=1091.447,35.993,-57.791,175.325,17.483,152.652
C07991=1091.453,36.243,-57.807,175.327,17.485,152.652
C07992=1091.458,36.492,-57.822,175.329,17.486,152.652
C07993=1091.464,36.742,-57.837,175.331,17.488,152.652
C07994=1091.470,36.990,-57.853,175.333,17.489,152.652
C07995=1091.476,37.240,-57.868,175.334,17.490,152.652
C07996=1091.482,37.490,-57.883,175.337,17.492,152.652
C07997=1091.487,37.739,-57.898,175.338,17.494,152.652
C07998=1091.493,37.989,-57.913,175.340,17.495,152.652
C07999=1091.499,38.238,-57.929,175.342,17.496,152.652
C08000=1091.504,38.487,-57.945,175.344,17.498,152.652
C08001=1091.510,38.737,-57.960,175.346,17.500,152.652
C08002=1091.515,38.986,-57.975,175.348,17.501,152.652
C08003=1091.521,39.236,-57.991,175.349,17.502,152.652
C08004=1091.527,39.486,-58.007,175.351,17.504,152.652
C08005=1091.533,39.735,-58.021,175.353,17.505,152.651
C08006=1091.538,39.985,-58.037,175.356,17.507,152.651
C08007=1091.544,40.233,-58.053,175.357,17.508,152.651
C08008=1091.549,40.483,-58.068,175.359,17.509,152.651
C08009=1091.556,40.733,-58.083,175.361,17.511,152.651
C08010=1091.561,40.982,-58.099,175.363,17.512,152.651
C08011=1091.567,41.232,-58.114,175.365,17.514,152.651
C08012=1091.572,41.482,-58.130,175.367,17.515,152.651
C08013=1091.579,41.730,-58.145,175.369,17.517,152.651
C08014=1091.584,41.980,-58.161,175.371,17.518,152.651
C08015=1091.590,42.230,-58.176,175.372,17.520,152.651
C08016=1091.595,42.478,-58.192,175.374,17.521,152.651
C08017=1091.601,42.728,-58.208,175.376,17.522,152.651
C08018=1091.607,42.978,-58.223,175.379,17.524,152.650
C08019=1091.613,43.227,-58.239,175.380,17.526,152.650
C08020=1091.618,43.477,-58.254,175.382,17.527,152.650
C08021=1091.624,43.727,-58.270,175.384,17.528,152.650
C08022=1091.629,43.975,-58.286,175.386,17.530,152.650
C08023=1091.635,44.225,-58.301,175.388,17.532,152.650
C08024=1091.641,44.475,-58.317,175.389,17.533,152.650
C08025=1091.646,44.724,-58.333,175.391,17.534,152.650
C08026=1091.653,44.973,-58.348,175.394,17.536,152.650
C08027=1091.658,45.223,-58.364,175.395,17.537,152.650
C08028=1091.663,45.472,-58.379,175.397,17.539,152.650
C08029=1091.669,45.721,-58.395,175.399,17.540,152.650
C08030=1091.675,45.971,-58.411,175.401,17.542,152.649
C08031=1091.680,46.220,-58.427,175.403,17.543,152.650
C08032=1091.686,46.470,-58.442,175.404,17.544,152.649
C08033=1091.692,46.719,-58.458,175.407,17.546,152.649
C08034=1091.697,46.969,-58.474,175.409,17.547,152.649
C08035=1091.703,47.245,-58.491,175.411,17.549,152.649
C08036=1091.710,47.522,-58.509,175.413,17.551,152.649
C08037=1091.716,47.798,-58.526,175.415,17.552,152.649
C08038=1091.722,48.075,-58.544,175.417,17.554,152.649
C08039=1091.727,48.323,-58.560,175.420,17.556,152.649
C08040=1091.733,48.573,-58.576,175.421,17.557,152.649
C08041=1091.738,48.823,-58.592,175.423,17.558,152.649
C08042=1091.744,49.072,-58.608,175.425,17.560,152.649
C08043=1091.749,49.321,-58.623,175.427,17.561,152.648
C08044=1091.755,49.571,-58.640,175.429,17.563,152.648
C08045=1091.761,49.821,-58.655,175.431,17.564,152.648
C08046=1091.767,50.070,-58.671,175.433,17.566,152.648
C08047=1091.772,50.319,-58.687,175.435,17.567,152.648
C08048=1091.778,50.569,-58.703,175.436,17.568,152.648
C08049=1091.784,50.818,-58.719,175.439,17.569,152.648
C08050=1091.790,51.067,-58.735,175.440,17.571,152.648
C08051=1091.795,51.317,-58.751,175.443,17.573,152.648
C08052=1091.801,51.566,-58.767,175.444,17.574,152.648
C08053=1091.807,51.815,-58.783,175.447,17.575,152.648
C08054=1091.812,52.065,-58.799,175.448,17.576,152.648
C08055=1091.818,52.314,-58.814,175.451,17.578,152.647
C08056=1091.824,52.563,-58.831,175.453,17.579,152.647
C08057=1091.829,52.813,-58.846,175.454,17.580,152.647
C08058=1091.835,53.063,-58.863,175.457,17.582,152.647
C08059=1091.841,53.312,-58.879,175.458,17.584,152.647
C08060=1091.846,53.562,-58.895,175.461,17.585,152.647
C08061=1091.852,53.811,-58.911,175.462,17.586,152.647
C08062=1091.858,54.060,-58.927,175.465,17.588,152.647
C08063=1091.863,54.310,-58.943,175.466,17.589,152.647
C08064=1091.869,54.560,-58.959,175.469,17.591,152.647
C08065=1091.875,54.809,-58.975,175.470,17.592,152.646
C08066=1091.881,55.058,-58.991,175.472,17.593,152.646
C08067=1091.886,55.307,-59.007,175.474,17.595,152.646
C08068=1091.892,55.556,-59.023,175.476,17.596,152.646
C08069=1091.897,55.807,-59.040,175.479,17.597,152.646
C08070=1091.903,56.056,-59.056,175.480,17.598,152.646
C08071=1091.909,56.305,-59.072,175.483,17.600,152.646
C08072=1091.915,56.555,-59.088,175.484,17.601,152.646
C08073=1091.921,56.804,-59.105,175.487,17.603,152.646
C08074=1091.927,57.054,-59.120,175.488,17.604,152.645
C08075=1091.932,57.303,-59.136,175.491,17.606,152.645
C08076=1091.938,57.552,-59.152,175.492,17.607,152.645
C08077=1091.943,57.802,-59.169,175.494,17.608,152.645
C08078=1091.949,58.051,-59.185,175.497,17.609,152.645
C08079=1091.955,58.300,-59.202,175.498,17.611,152.645
C08080=1091.961,58.550,-59.218,175.501,17.612,152.645
C08081=1091.967,58.799,-59.234,175.502,17.613,152.645
C08082=1091.973,59.048,-59.250,175.505,17.615,152.645
C08083=1091.978,59.299,-59.267,175.506,17.616,152.644
C08084=1091.984,59.548,-59.283,175.509,17.618,152.644
C08085=1091.990,59.797,-59.299,175.511,17.619,152.644
C08086=1091.996,60.047,-59.315,175.513,17.620,152.644
C08087=1092.002,60.296,-59.332,175.515,17.622,152.644
C08088=1092.007,60.545,-59.348,175.517,17.623,152.644
C08089=1092.012,60.794,-59.364,175.519,17.624,152.644
C08090=1092.018,61.044,-59.381,175.521,17.626,152.644
C08091=1092.024,61.293,-59.397,175.523,17.627,152.644
C08092=1092.030,61.542,-59.413,175.524,17.628,152.643
C08093=1092.036,61.792,-59.429,175.527,17.630,152.643
C08094=1092.041,62.041,-59.446,175.529,17.630,152.643
C08095=1092.047,62.291,-59.463,175.531,17.632,152.643
C08096=1092.053,62.540,-59.479,175.533,17.633,152.643
C08097=1092.059,62.789,-59.495,175.535,17.635,152.643
C08098=1092.064,63.039,-59.512,175.537,17.636,152.643
C08099=1092.071,63.315,-59.530,175.540,17.638,152.642
C08100=1092.078,63.591,-59.548,175.542,17.639,152.642
C08101=1092.084,63.867,-59.567,175.544,17.641,152.642
C08102=1092.091,64.144,-59.585,175.546,17.641,152.642
C08103=1092.096,64.393,-59.601,175.549,17.643,152.642
C08104=1092.103,64.642,-59.618,175.550,17.644,152.642
C08105=1092.108,64.892,-59.635,175.553,17.646,152.642
C08106=1092.114,65.141,-59.651,175.555,17.647,152.642
C08107=1092.120,65.390,-59.668,175.557,17.649,152.641
C08108=1092.125,65.640,-59.684,175.559,17.650,152.641
C08109=1092.130,65.889,-59.700,175.561,17.651,152.641
C08110=1092.136,66.138,-59.717,175.563,17.652,152.641
C08111=1092.142,66.388,-59.733,175.565,17.654,152.641
C08112=1092.148,66.637,-59.750,175.567,17.655,152.641
C08113=1092.154,66.887,-59.768,175.570,17.656,152.641
C08114=1092.160,67.136,-59.784,175.571,17.657,152.640
C08115=1092.165,67.386,-59.801,175.574,17.659,152.640
C08116=1092.171,67.635,-59.817,175.575,17.660,152.640
C08117=1092.176,67.884,-59.835,175.578,17.662,152.640
C08118=1092.182,68.134,-59.851,175.579,17.663,152.640
C08119=1092.187,68.383,-59.868,175.582,17.664,152.640
C08120=1092.193,68.633,-59.884,175.584,17.665,152.640
C08121=1092.199,68.882,-59.901,175.586,17.667,152.639
C08122=1092.205,69.131,-59.918,175.588,17.668,152.639
C08123=1092.210,69.381,-59.935,175.590,17.670,152.639
C08124=1092.216,69.630,-59.951,175.592,17.671,152.639
C08125=1092.222,69.879,-59.968,175.595,17.672,152.639
C08126=1092.228,70.128,-59.985,175.596,17.673,152.639
C08127=1092.233,70.378,-60.002,175.599,17.675,152.639
C08128=1092.239,70.627,-60.018,175.600,17.676,152.639
C08129=1092.244,70.876,-60.035,175.603,17.677,152.638
C08130=1092.250,71.126,-60.052,175.605,17.679,152.638
C08131=1092.255,71.375,-60.068,175.607,17.680,152.638
C08132=1092.261,71.625,-60.086,175.609,17.681,152.638
C08133=1092.267,71.874,-60.102,175.611,17.682,152.638
C08134=1092.272,72.124,-60.119,175.613,17.684,152.638
C08135=1092.278,72.372,-60.136,175.616,17.685,152.638
C08136=1092.284,72.623,-60.153,175.617,17.686,152.637
C08137=1092.290,72.872,-60.171,175.620,17.687,152.637
C08138=1092.296,73.121,-60.187,175.622,17.689,152.637
C08139=1092.301,73.371,-60.204,175.624,17.690,152.637
C08140=1092.306,73.620,-60.222,175.626,17.691,152.637
C08141=1092.312,73.869,-60.238,175.628,17.692,152.637
C08142=1092.318,74.118,-60.255,175.630,17.694,152.637
C08143=1092.324,74.367,-60.272,175.632,17.695,152.636
C08144=1092.329,74.617,-60.288,175.634,17.696,152.636
C08145=1092.334,74.866,-60.306,175.637,17.697,152.636
C08146=1092.341,75.116,-60.323,175.638,17.699,152.636
C08147=1092.347,75.365,-60.340,175.641,17.700,152.636
C08148=1092.352,75.615,-60.357,175.643,17.701,152.636
C08149=1092.358,75.864,-60.374,175.645,17.702,152.635
C08150=1092.363,76.113,-60.391,175.647,17.704,152.635
C08151=1092.369,76.362,-60.408,175.649,17.705,152.635
C08152=1092.375,76.612,-60.425,175.651,17.706,152.635
C08153=1092.381,76.861,-60.443,175.654,17.708,152.635
C08154=1092.386,77.111,-60.460,175.655,17.709,152.635
C08155=1092.392,77.360,-60.477,175.658,17.710,152.635
C08156=1092.397,77.609,-60.493,175.661,17.711,152.634
C08157=1092.403,77.858,-60.511,175.662,17.713,152.634
C08158=1092.409,78.108,-60.528,175.665,17.714,152.634
C08159=1092.415,78.358,-60.545,175.667,17.715,152.634
C08160=1092.421,78.607,-60.563,175.669,17.716,152.634
C08161=1092.426,78.856,-60.580,175.671,17.718,152.634
C08162=1092.431,79.105,-60.597,175.673,17.719,152.633
C08163=1092.437,79.381,-60.616,175.676,17.720,152.633
C08164=1092.443,79.657,-60.635,175.678,17.721,152.633
C08165=1092.450,79.934,-60.655,175.680,17.723,152.633
C08166=1092.456,80.210,-60.673,175.683,17.724,152.633
C08167=1092.462,80.459,-60.690,175.684,17.725,152.633
C08168=1092.468,80.708,-60.708,175.687,17.727,152.632
C08169=1092.473,80.957,-60.725,175.690,17.728,152.632
C08170=1092.478,81.206,-60.742,175.691,17.729,152.632
C08171=1092.485,81.456,-60.760,175.694,17.730,152.632
C08172=1092.490,81.706,-60.777,175.696,17.732,152.632
C08173=1092.495,81.955,-60.795,175.698,17.733,152.632
C08174=1092.501,82.204,-60.812,175.700,17.734,152.631
C08175=1092.506,82.453,-60.830,175.702,17.735,152.631
C08176=1092.513,82.703,-60.846,175.704,17.736,152.631
C08177=1092.518,82.952,-60.864,175.707,17.738,152.631
C08178=1092.524,83.201,-60.882,175.708,17.739,152.631
C08179=1092.529,83.451,-60.898,175.711,17.740,152.631
C08180=1092.535,83.701,-60.916,175.714,17.742,152.630
C08181=1092.541,83.950,-60.934,175.716,17.742,152.630
C08182=1092.546,84.199,-60.952,175.718,17.744,152.630
C08183=1092.552,84.448,-60.969,175.720,17.745,152.630
C08184=1092.558,84.698,-60.986,175.722,17.746,152.630
C08185=1092.563,84.947,-61.004,175.724,17.747,152.630
C08186=1092.569,85.196,-61.021,175.727,17.748,152.629
C08187=1092.574,85.445,-61.039,175.728,17.750,152.629
C08188=1092.580,85.695,-61.057,175.731,17.751,152.629
C08189=1092.586,85.945,-61.074,175.734,17.752,152.629
C08190=1092.591,86.194,-61.091,175.735,17.753,152.629
C08191=1092.597,86.443,-61.109,175.738,17.755,152.628
C08192=1092.603,86.692,-61.127,175.740,17.755,152.628
C08193=1092.609,86.941,-61.144,175.742,17.757,152.628
C08194=1092.614,87.190,-61.161,175.744,17.757,152.628
C08195=1092.621,87.440,-61.179,175.747,17.759,152.628
C08196=1092.626,87.689,-61.197,175.749,17.760,152.628
C08197=1092.632,87.938,-61.214,175.751,17.761,152.627
C08198=1092.637,88.188,-61.232,175.754,17.763,152.627
C08199=1092.643,88.437,-61.249,175.755,17.764,152.627
C08200=1092.648,88.686,-61.267,175.758,17.765,152.627
C08201=1092.655,88.936,-61.285,175.760,17.766,152.627
C08202=1092.660,89.185,-61.302,175.763,17.767,152.626
C08203=1092.666,89.434,-61.320,175.764,17.768,152.626
C08204=1092.672,89.684,-61.338,175.767,17.769,152.626
C08205=1092.677,89.933,-61.355,175.770,17.771,152.626
C08206=1092.682,90.182,-61.374,175.771,17.772,152.626
C08207=1092.688,90.432,-61.391,175.774,17.773,152.625
C08208=1092.694,90.681,-61.409,175.776,17.774,152.625
C08209=1092.700,90.931,-61.427,175.778,17.775,152.625
C08210=1092.705,91.180,-61.445,175.780,17.776,152.625
C08211=1092.711,91.429,-61.462,175.783,17.777,152.625
C08212=1092.717,91.679,-61.480,175.785,17.779,152.625
C08213=1092.722,91.928,-61.498,175.787,17.780,152.624
C08214=1092.727,92.177,-61.516,175.790,17.781,152.624
C08215=1092.734,92.426,-61.534,175.792,17.782,152.624
C08216=1092.739,92.675,-61.552,175.794,17.783,152.624
C08217=1092.745,92.924,-61.570,175.796,17.784,152.624
C08218=1092.751,93.174,-61.587,175.799,17.785,152.623
C08219=1092.756,93.423,-61.606,175.801,17.787,152.623
C08220=1092.761,93.672,-61.623,175.803,17.788,152.623
C08221=1092.767,93.922,-61.641,175.806,17.789,152.623
C08222=1092.773,94.171,-61.659,175.807,17.790,152.623
C08223=1092.778,94.420,-61.676,175.810,17.791,152.622
C08224=1092.784,94.670,-61.696,175.813,17.793,152.622
C08225=1092.790,94.919,-61.713,175.814,17.793,152.622
C08226=1092.796,95.168,-61.731,175.817,17.794,152.622
C08227=1092.801,95.444,-61.751,175.820,17.796,152.621
C08228=1092.808,95.721,-61.771,175.822,17.797,152.621
C08229=1092.814,95.996,-61.791,175.824,17.798,152.621
C08230=1092.820,96.273,-61.811,175.827,17.799,152.621
C08231=1092.826,96.522,-61.829,175.829,17.801,152.621
C08232=1092.832,96.771,-61.847,175.831,17.801,152.620
C08233=1092.837,97.021,-61.865,175.834,17.802,152.620
C08234=1092.843,97.270,-61.883,175.837,17.804,152.620
C08235=1092.849,97.519,-61.901,175.839,17.805,152.620
C08236=1092.854,97.769,-61.919,175.841,17.806,152.619
C08237=1092.860,98.018,-61.937,175.843,17.807,152.619
C08238=1092.865,98.266,-61.955,175.846,17.808,152.619
C08239=1092.871,98.516,-61.973,175.848,17.809,152.619
C08240=1092.876,98.765,-61.991,175.850,17.810,152.619
C08241=1092.883,99.015,-62.010,175.853,17.812,152.618
C08242=1092.888,99.264,-62.028,175.855,17.812,152.618
C08243=1092.894,99.514,-62.046,175.857,17.813,152.618
C08244=1092.899,99.762,-62.064,175.860,17.815,152.618
C08245=1092.906,100.012,-62.082,175.862,17.816,152.618
C08246=1092.910,100.261,-62.101,175.864,17.817,152.617
C08247=1092.917,100.510,-62.119,175.866,17.817,152.617
C08248=1092.922,100.759,-62.137,175.869,17.819,152.617
C08249=1092.928,101.009,-62.156,175.872,17.820,152.616
C08250=1092.933,101.258,-62.174,175.873,17.821,152.616
C08251=1092.940,101.508,-62.191,175.876,17.822,152.616
C08252=1092.945,101.756,-62.210,175.878,17.823,152.616
C08253=1092.951,102.006,-62.228,175.881,17.824,152.616
C08254=1092.956,102.255,-62.247,175.883,17.825,152.615
C08255=1092.962,102.505,-62.265,175.885,17.826,152.615
C08256=1092.967,102.754,-62.283,175.888,17.827,152.615
C08257=1092.973,103.003,-62.302,175.890,17.828,152.615
C08258=1092.978,103.252,-62.320,175.892,17.830,152.615
C08259=1092.984,103.501,-62.339,175.895,17.831,152.614
C08260=1092.989,103.751,-62.357,175.897,17.831,152.614
C08261=1092.996,104.000,-62.376,175.900,17.832,152.614
C08262=1093.000,104.249,-62.394,175.902,17.834,152.614
C08263=1093.007,104.498,-62.412,175.904,17.835,152.613
C08264=1093.012,104.748,-62.430,175.907,17.836,152.613
C08265=1093.017,104.997,-62.450,175.909,17.837,152.613
C08266=1093.023,105.246,-62.467,175.911,17.838,152.613
C08267=1093.029,105.496,-62.487,175.914,17.839,152.612
C08268=1093.035,105.745,-62.505,175.916,17.839,152.612
C08269=1093.040,105.994,-62.523,175.919,17.841,152.612
C08270=1093.046,106.243,-62.542,175.921,17.842,152.612
C08271=1093.051,106.493,-62.560,175.923,17.843,152.612
C08272=1093.057,106.742,-62.579,175.926,17.844,152.611
C08273=1093.062,106.991,-62.597,175.928,17.845,152.611
C08274=1093.068,107.241,-62.616,175.931,17.846,152.611
C08275=1093.074,107.490,-62.635,175.933,17.847,152.610
C08276=1093.079,107.739,-62.653,175.935,17.848,152.610
C08277=1093.085,107.988,-62.672,175.938,17.849,152.610
C08278=1093.091,108.237,-62.691,175.941,17.850,152.610
C08279=1093.097,108.487,-62.708,175.943,17.851,152.609
C08280=1093.102,108.736,-62.728,175.945,17.852,152.609
C08281=1093.107,108.985,-62.747,175.948,17.853,152.609
C08282=1093.114,109.235,-62.765,175.950,17.854,152.609
C08283=1093.119,109.484,-62.784,175.952,17.855,152.609
C08284=1093.125,109.732,-62.802,175.954,17.856,152.608
C08285=1093.131,109.982,-62.821,175.957,17.857,152.608
C08286=1093.136,110.231,-62.839,175.960,17.858,152.608
C08287=1093.142,110.480,-62.858,175.962,17.859,152.608
C08288=1093.148,110.730,-62.877,175.964,17.860,152.607
C08289=1093.153,110.978,-62.896,175.967,17.861,152.607
C08290=1093.159,111.228,-62.914,175.969,17.862,152.607
C08291=1093.165,111.504,-62.935,175.972,17.862,152.606
C08292=1093.171,111.781,-62.956,175.975,17.864,152.606
C08293=1093.178,112.057,-62.977,175.977,17.865,152.606
C08294=1093.184,112.333,-62.998,175.980,17.866,152.605
C08295=1093.189,112.582,-63.016,175.983,17.867,152.605
C08296=1093.195,112.831,-63.036,175.985,17.868,152.605
C08297=1093.201,113.080,-63.054,175.988,17.869,152.605
C08298=1093.207,113.330,-63.074,175.990,17.870,152.604
C08299=1093.212,113.579,-63.092,175.992,17.871,152.604
C08300=1093.218,113.828,-63.112,175.995,17.872,152.604
C08301=1093.224,114.078,-63.130,175.998,17.873,152.604
C08302=1093.229,114.326,-63.148,176.000,17.874,152.603
C08303=1093.234,114.576,-63.168,176.002,17.875,152.603
C08304=1093.240,114.825,-63.187,176.005,17.876,152.603
C08305=1093.245,115.074,-63.206,176.007,17.877,152.603
C08306=1093.251,115.324,-63.225,176.010,17.878,152.602
C08307=1093.257,115.573,-63.244,176.012,17.879,152.602
C08308=1093.262,115.821,-63.263,176.014,17.880,152.602
C08309=1093.268,116.071,-63.282,176.017,17.881,152.602
C08310=1093.274,116.320,-63.301,176.020,17.882,152.601
C08311=1093.279,116.569,-63.320,176.022,17.883,152.601
C08312=1093.285,116.818,-63.339,176.024,17.884,152.601
C08313=1093.290,117.068,-63.358,176.027,17.885,152.601
C08314=1093.295,117.317,-63.377,176.029,17.886,152.600
C08315=1093.301,117.566,-63.397,176.032,17.887,152.600
C08316=1093.307,117.815,-63.416,176.035,17.887,152.600
C08317=1093.312,118.064,-63.435,176.037,17.888,152.599
C08318=1093.317,118.314,-63.454,176.039,17.889,152.599
C08319=1093.323,118.563,-63.473,176.042,17.890,152.599
C08320=1093.329,118.812,-63.492,176.044,17.891,152.599
C08321=1093.334,119.061,-63.511,176.047,17.892,152.598
C08322=1093.340,119.311,-63.531,176.050,17.893,152.598
C08323=1093.345,119.560,-63.550,176.051,17.894,152.598
C08324=1093.351,119.809,-63.569,176.054,17.895,152.598
C08325=1093.356,120.058,-63.588,176.057,17.896,152.597
C08326=1093.362,120.308,-63.607,176.059,17.896,152.597
C08327=1093.367,120.557,-63.626,176.062,17.898,152.597
C08328=1093.373,120.807,-63.646,176.065,17.899,152.596
C08329=1093.379,121.055,-63.665,176.066,17.899,152.596
C08330=1093.384,121.304,-63.685,176.069,17.901,152.596
C08331=1093.390,121.553,-63.704,176.072,17.901,152.595
C08332=1093.396,121.803,-63.723,176.074,17.902,152.595
C08333=1093.401,122.052,-63.742,176.077,17.903,152.595
C08334=1093.406,122.301,-63.761,176.080,17.904,152.595
C08335=1093.412,122.550,-63.781,176.081,17.905,152.594
C08336=1093.418,122.799,-63.800,176.084,17.906,152.594
C08337=1093.424,123.049,-63.820,176.087,17.907,152.594
C08338=1093.429,123.298,-63.839,176.090,17.908,152.593
C08339=1093.435,123.547,-63.858,176.092,17.909,152.593
C08340=1093.441,123.796,-63.878,176.095,17.909,152.593
C08341=1093.446,124.045,-63.897,176.098,17.910,152.593
C08342=1093.452,124.295,-63.916,176.099,17.911,152.592
C08343=1093.458,124.544,-63.935,176.102,17.912,152.592
C08344=1093.464,124.793,-63.955,176.105,17.913,152.592
C08345=1093.469,125.043,-63.975,176.107,17.914,152.591
C08346=1093.474,125.291,-63.994,176.110,17.915,152.591
C08347=1093.480,125.540,-64.014,176.113,17.915,152.591
C08348=1093.485,125.790,-64.033,176.115,17.916,152.590
C08349=1093.491,126.039,-64.052,176.117,17.917,152.590
C08350=1093.497,126.288,-64.072,176.120,17.918,152.590
C08351=1093.503,126.537,-64.092,176.123,17.919,152.589
C08352=1093.508,126.787,-64.111,176.125,17.920,152.589
C08353=1093.514,127.035,-64.131,176.128,17.920,152.589
C08354=1093.520,127.285,-64.150,176.131,17.922,152.589
C08355=1093.526,127.561,-64.172,176.134,17.922,152.588
C08356=1093.532,127.836,-64.194,176.136,17.923,152.588
C08357=1093.538,128.113,-64.216,176.139,17.924,152.587
C08358=1093.545,128.389,-64.237,176.142,17.925,152.587
C08359=1093.550,128.638,-64.256,176.144,17.925,152.587
C08360=1093.556,128.887,-64.276,176.147,17.927,152.587
C08361=1093.561,129.137,-64.296,176.150,17.927,152.586
C08362=1093.567,129.385,-64.316,176.152,17.928,152.586
C08363=1093.573,129.635,-64.335,176.155,17.929,152.585
C08364=1093.579,129.884,-64.355,176.158,17.930,152.585
C08365=1093.584,130.133,-64.374,176.161,17.931,152.585
C08366=1093.590,130.382,-64.394,176.163,17.931,152.585
C08367=1093.595,130.632,-64.414,176.165,17.932,152.584
C08368=1093.601,130.880,-64.434,176.168,17.933,152.584
C08369=1093.607,131.130,-64.453,176.170,17.934,152.584
C08370=1093.613,131.379,-64.473,176.173,17.934,152.583
C08371=1093.619,131.628,-64.492,176.176,17.936,152.583
C08372=1093.625,131.877,-64.512,176.179,17.936,152.583
C08373=1093.630,132.126,-64.533,176.181,17.936,152.582
C08374=1093.636,132.376,-64.552,176.184,17.938,152.582
C08375=1093.642,132.624,-64.572,176.187,17.939,152.582
C08376=1093.647,132.874,-64.592,176.189,17.939,152.581
C08377=1093.653,133.123,-64.612,176.192,17.940,152.581
C08378=1093.659,133.372,-64.632,176.195,17.941,152.581
C08379=1093.664,133.621,-64.652,176.197,17.942,152.580
C08380=1093.670,133.870,-64.672,176.199,17.942,152.580
C08381=1093.675,134.119,-64.692,176.202,17.943,152.580
C08382=1093.681,134.369,-64.712,176.205,17.944,152.579
C08383=1093.687,134.618,-64.732,176.208,17.945,152.579
C08384=1093.692,134.867,-64.752,176.210,17.945,152.579
C08385=1093.697,135.116,-64.771,176.213,17.946,152.578
C08386=1093.703,135.365,-64.792,176.216,17.947,152.578
C08387=1093.709,135.614,-64.812,176.219,17.948,152.578
C08388=1093.714,135.864,-64.831,176.221,17.948,152.577
C08389=1093.720,136.113,-64.852,176.223,17.950,152.577
C08390=1093.726,136.362,-64.872,176.226,17.950,152.577
C08391=1093.733,136.697,-64.898,176.229,17.951,152.576
C08392=1093.741,137.031,-64.925,176.233,17.952,152.576
C08393=1093.748,137.366,-64.953,176.237,17.954,152.575
C08394=1093.756,137.701,-64.980,176.240,17.954,152.575
C08395=1093.762,137.950,-65.000,176.243,17.955,152.574
C08396=1093.767,138.199,-65.020,176.246,17.956,152.574
C08397=1093.773,138.448,-65.040,176.249,17.957,152.574
C08398=1093.778,138.697,-65.061,176.251,17.957,152.573
C08399=1093.784,138.946,-65.080,176.254,17.958,152.573
C08400=1093.789,139.195,-65.100,176.257,17.959,152.573
C08401=1093.795,139.444,-65.120,176.260,17.960,152.572
C08402=1093.800,139.693,-65.141,176.262,17.960,152.572
C08403=1093.806,139.942,-65.161,176.265,17.961,152.572
C08404=1093.812,140.191,-65.181,176.268,17.962,152.571
C08405=1093.818,140.440,-65.201,176.270,17.963,152.571
C08406=1093.823,140.690,-65.222,176.272,17.963,152.571
C08407=1093.829,140.939,-65.242,176.275,17.964,152.570
C08408=1093.834,141.189,-65.262,176.278,17.965,152.570
C08409=1093.840,141.438,-65.283,176.281,17.966,152.569
C08410=1093.846,141.686,-65.303,176.284,17.967,152.569
C08411=1093.851,141.936,-65.323,176.286,17.967,152.569
C08412=1093.856,142.185,-65.344,176.289,17.968,152.568
C08413=1093.862,142.434,-65.364,176.292,17.969,152.568
C08414=1093.867,142.683,-65.384,176.295,17.969,152.568
C08415=1093.873,142.902,-65.402,176.297,17.970,152.567
C08416=1093.877,143.122,-65.420,176.299,17.970,152.567
C08417=1093.883,143.342,-65.438,176.302,17.971,152.567
C08418=1093.887,143.562,-65.456,176.304,17.972,152.566
C08419=1093.892,143.781,-65.475,176.306,17.973,152.566
C08420=1093.897,144.001,-65.493,176.309,17.973,152.566
C08421=1093.902,144.221,-65.511,176.311,17.974,152.566
C08422=1093.907,144.441,-65.529,176.314,17.974,152.565
C08423=1093.913,144.691,-65.549,176.317,17.975,152.565
C08424=1093.919,144.940,-65.569,176.319,17.976,152.564
C08425=1093.924,145.189,-65.590,176.321,17.976,152.564
C08426=1093.930,145.437,-65.611,176.324,17.977,152.564
C08427=1093.935,145.686,-65.631,176.327,17.978,152.563
C08428=1093.941,145.935,-65.652,176.330,17.978,152.563
C08429=1093.947,146.185,-65.672,176.333,17.980,152.563
C08430=1093.952,146.434,-65.693,176.335,17.980,152.562
C08431=1093.958,146.683,-65.713,176.338,17.980,152.562
C08432=1093.963,146.932,-65.734,176.341,17.981,152.561
C08433=1093.970,147.181,-65.755,176.344,17.982,152.561
C08434=1093.975,147.430,-65.775,176.346,17.983,152.561
C08435=1093.980,147.679,-65.796,176.349,17.983,152.560
C08436=1093.986,147.928,-65.817,176.352,17.984,152.560
C08437=1093.992,148.177,-65.836,176.355,17.985,152.559
C08438=1093.998,148.426,-65.858,176.358,17.985,152.559
C08439=1094.003,148.676,-65.879,176.360,17.985,152.559
C08440=1094.008,148.925,-65.899,176.363,17.987,152.558
C08441=1094.014,149.174,-65.920,176.366,17.987,152.558
C08442=1094.020,149.423,-65.941,176.369,17.988,152.558
C08443=1094.026,149.672,-65.961,176.372,17.989,152.557
C08444=1094.031,149.921,-65.982,176.374,17.989,152.557
C08445=1094.036,150.170,-66.002,176.377,17.990,152.556
C08446=1094.042,150.419,-66.024,176.380,17.991,152.556
C08447=1094.048,150.668,-66.045,176.383,17.992,152.556
C08448=1094.053,150.917,-66.065,176.386,17.992,152.555
C08449=1094.058,151.166,-66.086,176.388,17.992,152.555
C08450=1094.065,151.415,-66.107,176.391,17.993,152.555
C08451=1094.070,151.665,-66.127,176.394,17.994,152.554
C08452=1094.076,151.913,-66.149,176.397,17.995,152.554
C08453=1094.081,152.162,-66.169,176.400,17.996,152.553
C08454=1094.087,152.412,-66.190,176.402,17.996,152.553
C08455=1094.093,152.661,-66.211,176.405,17.997,152.553
C08456=1094.098,152.910,-66.232,176.408,17.997,152.552
C08457=1094.104,153.159,-66.254,176.411,17.998,152.552
C08458=1094.109,153.408,-66.274,176.414,17.999,152.551
C08459=1094.115,153.657,-66.295,176.416,17.999,152.551
C08460=1094.120,153.906,-66.316,176.419,18.000,152.551
C08461=1094.126,154.155,-66.337,176.422,18.000,152.550
C08462=1094.131,154.404,-66.358,176.425,18.001,152.550
C08463=1094.137,154.653,-66.379,176.428,18.002,152.549
C08464=1094.143,154.902,-66.400,176.431,18.003,152.549
C08465=1094.148,155.151,-66.421,176.433,18.003,152.549
C08466=1094.154,155.400,-66.442,176.436,18.003,152.548
C08467=1094.160,155.650,-66.463,176.439,18.004,152.548
C08468=1094.165,155.898,-66.484,176.442,18.005,152.547
C08469=1094.170,156.147,-66.505,176.445,18.006,152.547
C08470=1094.177,156.397,-66.527,176.447,18.006,152.547
C08471=1094.182,156.645,-66.548,176.450,18.006,152.546
C08472=1094.188,156.895,-66.569,176.453,18.007,152.546
C08473=1094.194,157.143,-66.590,176.456,18.008,152.545
C08474=1094.199,157.393,-66.611,176.459,18.009,152.545
C08475=1094.205,157.642,-66.632,176.462,18.009,152.544
C08476=1094.210,157.891,-66.653,176.464,18.009,152.544
C08477=1094.215,158.140,-66.675,176.467,18.010,152.544
C08478=1094.221,158.389,-66.696,176.470,18.011,152.543
C08479=1094.226,158.638,-66.717,176.473,18.012,152.543
C08480=1094.233,158.887,-66.738,176.476,18.012,152.542
C08481=1094.238,159.136,-66.760,176.479,18.013,152.542
C08482=1094.243,159.385,-66.780,176.482,18.013,152.542
C08483=1094.250,159.661,-66.804,176.485,18.014,152.541
C08484=1094.256,159.937,-66.828,176.489,18.015,152.541
C08485=1094.262,160.212,-66.852,176.492,18.015,152.540
C08486=1094.269,160.488,-66.875,176.495,18.016,152.540
C08487=1094.274,160.737,-66.896,176.498,18.017,152.539
C08488=1094.280,160.986,-66.918,176.501,18.018,152.539
C08489=1094.285,161.235,-66.939,176.503,18.017,152.539
C08490=1094.291,161.485,-66.960,176.506,18.018,152.538
C08491=1094.297,161.733,-66.982,176.509,18.019,152.538
C08492=1094.302,161.982,-67.003,176.512,18.019,152.537
C08493=1094.308,162.231,-67.025,176.515,18.020,152.537
C08494=1094.313,162.480,-67.046,176.518,18.021,152.536
C08495=1094.319,162.729,-67.067,176.521,18.022,152.536
C08496=1094.324,162.978,-67.089,176.523,18.022,152.536
C08497=1094.329,163.227,-67.110,176.526,18.022,152.535
C08498=1094.335,163.476,-67.133,176.529,18.023,152.535
C08499=1094.340,163.725,-67.154,176.532,18.024,152.534
C08500=1094.346,163.975,-67.175,176.535,18.025,152.534
C08501=1094.351,164.223,-67.197,176.538,18.025,152.534
C08502=1094.357,164.472,-67.218,176.541,18.026,152.533
C08503=1094.362,164.721,-67.240,176.544,18.027,152.533
C08504=1094.368,164.970,-67.262,176.546,18.027,152.532
C08505=1094.373,165.219,-67.284,176.549,18.028,152.532
C08506=1094.379,165.468,-67.305,176.552,18.028,152.532
C08507=1094.385,165.717,-67.327,176.555,18.029,152.531
C08508=1094.390,165.966,-67.349,176.558,18.029,152.531
C08509=1094.396,166.215,-67.370,176.561,18.030,152.530
C08510=1094.400,166.464,-67.392,176.564,18.031,152.530
C08511=1094.406,166.712,-67.413,176.567,18.031,152.529
C08512=1094.411,166.962,-67.436,176.570,18.032,152.529
C08513=1094.417,167.210,-67.457,176.573,18.032,152.529
C08514=1094.422,167.460,-67.479,176.576,18.033,152.528
C08515=1094.428,167.709,-67.500,176.579,18.033,152.528
C08516=1094.433,167.958,-67.523,176.582,18.034,152.527
C08517=1094.439,168.207,-67.544,176.585,18.035,152.527
C08518=1094.444,168.456,-67.566,176.588,18.036,152.526
C08519=1094.450,168.705,-67.587,176.591,18.036,152.526
C08520=1094.455,168.954,-67.610,176.593,18.036,152.526
C08521=1094.462,169.203,-67.631,176.596,18.037,152.525
C08522=1094.466,169.452,-67.653,176.599,18.037,152.525
C08523=1094.473,169.701,-67.675,176.602,18.038,152.524
C08524=1094.477,169.950,-67.697,176.605,18.038,152.524
C08525=1094.484,170.199,-67.718,176.608,18.039,152.523
C08526=1094.488,170.448,-67.740,176.611,18.040,152.523
C08527=1094.495,170.697,-67.762,176.614,18.041,152.523
C08528=1094.500,170.946,-67.784,176.618,18.041,152.522
C08529=1094.506,171.195,-67.806,176.620,18.041,152.522
C08530=1094.511,171.444,-67.828,176.623,18.042,152.521
C08531=1094.517,171.693,-67.849,176.626,18.042,152.521
C08532=1094.523,171.942,-67.872,176.629,18.043,152.520
C08533=1094.527,172.190,-67.894,176.632,18.043,152.520
C08534=1094.534,172.440,-67.916,176.635,18.044,152.519
C08535=1094.539,172.689,-67.938,176.638,18.044,152.519
C08536=1094.545,172.938,-67.959,176.641,18.045,152.518
C08537=1094.550,173.187,-67.982,176.644,18.046,152.518
C08538=1094.556,173.436,-68.004,176.647,18.046,152.518
C08539=1094.561,173.685,-68.026,176.650,18.046,152.517
C08540=1094.567,173.934,-68.049,176.653,18.047,152.517
C08541=1094.573,174.182,-68.070,176.656,18.047,152.516
C08542=1094.578,174.432,-68.092,176.659,18.048,152.516
C08543=1094.584,174.681,-68.114,176.662,18.048,152.515
C08544=1094.589,174.929,-68.136,176.665,18.049,152.515
C08545=1094.595,175.178,-68.159,176.668,18.050,152.514
C08546=1094.601,175.427,-68.181,176.671,18.050,152.514
C08547=1094.607,175.703,-68.205,176.674,18.051,152.513
C08548=1094.613,175.978,-68.230,176.678,18.051,152.513
C08549=1094.620,176.253,-68.255,176.681,18.051,152.512
C08550=1094.626,176.529,-68.279,176.685,18.053,152.512
C08551=1094.631,176.777,-68.301,176.688,18.053,152.511
C08552=1094.637,177.027,-68.323,176.690,18.053,152.511
C08553=1094.642,177.276,-68.345,176.693,18.053,152.510
C08554=1094.648,177.525,-68.368,176.696,18.054,152.510
C08555=1094.654,177.773,-68.389,176.700,18.054,152.509
C08556=1094.659,178.022,-68.412,176.703,18.055,152.509
C08557=1094.665,178.272,-68.435,176.706,18.055,152.508
C08558=1094.671,178.520,-68.457,176.709,18.056,152.508
C08559=1094.676,178.769,-68.479,176.712,18.056,152.507
C08560=1094.682,179.018,-68.502,176.715,18.057,152.507
C08561=1094.688,179.267,-68.523,176.718,18.057,152.507
C08562=1094.694,179.516,-68.546,176.721,18.058,152.506
C08563=1094.699,179.765,-68.568,176.725,18.058,152.506
C08564=1094.705,180.014,-68.591,176.728,18.059,152.505
C08565=1094.711,180.263,-68.614,176.730,18.059,152.505
C08566=1094.716,180.512,-68.636,176.733,18.059,152.504
C08567=1094.722,180.761,-68.659,176.736,18.060,152.504
C08568=1094.728,181.009,-68.680,176.739,18.060,152.503
C08569=1094.733,181.258,-68.703,176.742,18.061,152.503
C08570=1094.739,181.507,-68.726,176.746,18.061,152.502
C08571=1094.745,181.756,-68.748,176.749,18.062,152.502
C08572=1094.751,182.005,-68.770,176.752,18.062,152.501
C08573=1094.757,182.254,-68.793,176.755,18.062,152.501
C08574=1094.762,182.504,-68.816,176.758,18.063,152.500
C08575=1094.768,182.752,-68.838,176.761,18.063,152.500
C08576=1094.774,183.001,-68.861,176.764,18.064,152.499
C08577=1094.779,183.250,-68.883,176.768,18.064,152.499
C08578=1094.785,183.499,-68.906,176.771,18.064,152.498
C08579=1094.791,183.748,-68.929,176.774,18.065,152.498
C08580=1094.797,183.996,-68.951,176.777,18.065,152.497
C08581=1094.802,184.246,-68.973,176.780,18.065,152.497
C08582=1094.808,184.495,-68.996,176.783,18.066,152.496
C08583=1094.813,184.743,-69.019,176.786,18.066,152.496
C08584=1094.820,184.992,-69.041,176.789,18.066,152.495
C08585=1094.825,185.241,-69.063,176.792,18.067,152.495
C08586=1094.831,185.490,-69.086,176.795,18.067,152.494
C08587=1094.836,185.739,-69.110,176.798,18.068,152.494
C08588=1094.842,185.988,-69.133,176.802,18.068,152.493
C08589=1094.847,186.236,-69.155,176.805,18.069,152.493
C08590=1094.852,186.486,-69.178,176.808,18.070,152.492
C08591=1094.858,186.735,-69.201,176.811,18.070,152.492
C08592=1094.864,186.984,-69.224,176.814,18.071,152.491
C08593=1094.869,187.233,-69.246,176.817,18.071,152.491
C08594=1094.875,187.481,-69.269,176.820,18.072,152.490
C08595=1094.880,187.730,-69.292,176.823,18.072,152.490
C08596=1094.885,187.979,-69.316,176.826,18.073,152.489
C08597=1094.891,188.228,-69.338,176.829,18.073,152.489
C08598=1094.896,188.477,-69.361,176.833,18.074,152.489
C08599=1094.902,188.726,-69.384,176.836,18.074,152.488
C08600=1094.908,188.975,-69.407,176.839,18.075,152.488
C08601=1094.913,189.223,-69.429,176.842,18.075,152.487
C08602=1094.919,189.472,-69.452,176.845,18.076,152.487
C08603=1094.924,189.721,-69.476,176.848,18.076,152.486
C08604=1094.929,189.970,-69.499,176.852,18.076,152.486
C08605=1094.935,190.219,-69.522,176.855,18.077,152.485
C08606=1094.941,190.468,-69.545,176.858,18.077,152.485
C08607=1094.947,190.717,-69.567,176.861,18.078,152.484
C08608=1094.952,190.966,-69.591,176.864,18.078,152.484
C08609=1094.957,191.215,-69.614,176.867,18.078,152.483
C08610=1094.962,191.463,-69.637,176.870,18.079,152.483
C08611=1094.969,191.738,-69.662,176.874,18.079,152.482
C08612=1094.975,192.013,-69.688,176.877,18.080,152.482
C08613=1094.982,192.288,-69.713,176.881,18.081,152.481
C08614=1094.988,192.564,-69.739,176.884,18.081,152.480
C08615=1094.993,192.812,-69.762,176.887,18.081,152.480
C08616=1094.999,193.061,-69.785,176.890,18.082,152.479
C08617=1095.004,193.311,-69.809,176.894,18.082,152.479
C08618=1095.010,193.559,-69.832,176.897,18.082,152.478
C08619=1095.016,193.808,-69.855,176.900,18.083,152.478
C08620=1095.022,194.057,-69.878,176.903,18.083,152.477
C08621=1095.027,194.306,-69.902,176.906,18.084,152.477
C08622=1095.032,194.555,-69.925,176.910,18.084,152.476
C08623=1095.038,194.804,-69.948,176.913,18.085,152.476
C08624=1095.044,195.053,-69.971,176.916,18.085,152.475
C08625=1095.049,195.301,-69.995,176.919,18.085,152.475
C08626=1095.055,195.550,-70.018,176.922,18.086,152.474
C08627=1095.061,195.799,-70.041,176.925,18.086,152.474
C08628=1095.066,196.048,-70.064,176.929,18.087,152.473
C08629=1095.072,196.296,-70.088,176.932,18.087,152.473
C08630=1095.077,196.545,-70.111,176.935,18.087,152.472
C08631=1095.083,196.794,-70.134,176.938,18.088,152.472
C08632=1095.088,197.043,-70.158,176.941,18.088,152.471
C08633=1095.094,197.292,-70.181,176.945,18.089,152.471
C08634=1095.100,197.541,-70.204,176.948,18.089,152.470
C08635=1095.105,197.789,-70.228,176.951,18.089,152.470
C08636=1095.111,198.038,-70.251,176.954,18.089,152.469
C08637=1095.117,198.287,-70.274,176.957,18.090,152.469
C08638=1095.122,198.536,-70.299,176.961,18.090,152.468
C08639=1095.128,198.785,-70.322,176.964,18.091,152.468
C08640=1095.134,199.033,-70.346,176.967,18.091,152.467
C08641=1095.139,199.283,-70.369,176.970,18.091,152.467
C08642=1095.145,199.531,-70.392,176.974,18.092,152.466
C08643=1095.151,199.780,-70.416,176.977,18.092,152.465
C08644=1095.156,200.029,-70.439,176.981,18.093,152.465
C08645=1095.162,200.277,-70.463,176.984,18.094,152.464
C08646=1095.168,200.526,-70.486,176.987,18.094,152.464
C08647=1095.174,200.775,-70.511,176.990,18.094,152.463
C08648=1095.179,201.024,-70.533,176.994,18.094,152.463
C08649=1095.185,201.273,-70.558,176.997,18.095,152.462
C08650=1095.190,201.522,-70.581,177.000,18.095,152.462
C08651=1095.197,201.770,-70.604,177.003,18.095,152.461
C08652=1095.202,202.019,-70.628,177.007,18.096,152.461
C08653=1095.208,202.268,-70.652,177.010,18.096,152.460
C08654=1095.213,202.517,-70.675,177.013,18.097,152.460
C08655=1095.219,202.766,-70.699,177.016,18.097,152.459
C08656=1095.224,203.014,-70.723,177.019,18.097,152.459
C08657=1095.230,203.263,-70.746,177.022,18.097,152.458
C08658=1095.236,203.512,-70.771,177.026,18.098,152.457
C08659=1095.242,203.761,-70.794,177.029,18.098,152.457
C08660=1095.247,204.010,-70.818,177.032,18.098,152.456
C08661=1095.252,204.259,-70.842,177.035,18.099,152.456
C08662=1095.258,204.508,-70.865,177.038,18.099,152.455
C08663=1095.263,204.756,-70.890,177.042,18.100,152.455
C08664=1095.269,205.004,-70.913,177.046,18.101,152.454
C08665=1095.275,205.254,-70.937,177.049,18.101,152.454
C08666=1095.280,205.503,-70.961,177.052,18.101,152.453
C08667=1095.286,205.751,-70.985,177.055,18.101,152.453
C08668=1095.292,206.000,-71.009,177.058,18.102,152.452
C08669=1095.297,206.249,-71.033,177.062,18.102,152.452
C08670=1095.303,206.498,-71.057,177.065,18.103,152.451
C08671=1095.309,206.747,-71.081,177.068,18.103,152.451
C08672=1095.314,206.995,-71.105,177.071,18.103,152.450
C08673=1095.320,207.244,-71.128,177.075,18.104,152.450
C08674=1095.326,207.493,-71.153,177.078,18.104,152.449
C08675=1095.348,208.507,-71.251,177.131,18.126,152.444
C08676=1095.357,208.881,-71.287,177.136,18.128,152.443
C08677=1095.365,209.255,-71.324,177.140,18.130,152.443
C08678=1095.374,209.629,-71.360,177.145,18.132,152.443
C08679=1095.382,210.002,-71.398,177.150,18.134,152.442
C08680=1095.388,210.251,-71.422,177.153,18.135,152.442
C08681=1095.394,210.500,-71.446,177.156,18.137,152.441
C08682=1095.399,210.748,-71.470,177.159,18.138,152.441
C08683=1095.405,210.998,-71.495,177.162,18.139,152.441
C08684=1095.410,211.246,-71.519,177.165,18.140,152.441
C08685=1095.416,211.495,-71.543,177.168,18.141,152.440
C08686=1095.421,211.744,-71.568,177.172,18.143,152.440
C08687=1095.427,211.993,-71.592,177.174,18.144,152.440
C08688=1095.433,212.241,-71.617,177.177,18.145,152.439
C08689=1095.438,212.490,-71.642,177.181,18.147,152.439
C08690=1095.444,212.738,-71.666,177.184,18.148,152.439
C08691=1095.449,212.988,-71.691,177.187,18.149,152.438
C08692=1095.455,213.236,-71.715,177.190,18.151,152.438
C08693=1095.461,213.485,-71.740,177.193,18.151,152.438
C08694=1095.466,213.734,-71.764,177.197,18.153,152.437
C08695=1095.472,213.982,-71.789,177.200,18.154,152.437
C08696=1095.477,214.231,-71.813,177.202,18.155,152.437
C08697=1095.483,214.479,-71.838,177.206,18.157,152.437
C08698=1095.489,214.729,-71.863,177.209,18.158,152.436
C08699=1095.494,214.977,-71.887,177.212,18.159,152.436
C08700=1095.500,215.226,-71.913,177.215,18.161,152.436
C08701=1095.505,215.475,-71.937,177.218,18.161,152.435
C08702=1095.510,215.723,-71.962,177.222,18.163,152.435
C08703=1095.517,215.972,-71.987,177.224,18.165,152.435
C08704=1095.522,216.221,-72.011,177.228,18.166,152.434
C08705=1095.528,216.470,-72.036,177.231,18.167,152.434
C08706=1095.533,216.718,-72.061,177.235,18.168,152.434
C08707=1095.539,216.967,-72.085,177.237,18.170,152.433
C08708=1095.544,217.216,-72.111,177.240,18.171,152.433
C08709=1095.550,217.465,-72.136,177.244,18.172,152.433
C08710=1095.556,217.713,-72.161,177.247,18.173,152.433
C08711=1095.562,217.962,-72.185,177.250,18.175,152.432
C08712=1095.567,218.211,-72.209,177.253,18.176,152.432
C08713=1095.573,218.459,-72.235,177.256,18.177,152.432
C08714=1095.578,218.708,-72.260,177.260,18.179,152.431
C08715=1095.584,218.957,-72.285,177.262,18.180,152.431
C08716=1095.589,219.205,-72.309,177.266,18.182,152.431
C08717=1095.595,219.454,-72.335,177.269,18.182,152.430
C08718=1095.601,219.702,-72.359,177.272,18.184,152.430
C08719=1095.606,219.952,-72.385,177.275,18.185,152.430
C08720=1095.612,220.200,-72.410,177.278,18.186,152.429
C08721=1095.618,220.449,-72.434,177.282,18.188,152.429
C08722=1095.624,220.698,-72.460,177.285,18.189,152.429
C08723=1095.628,220.947,-72.484,177.288,18.191,152.429
C08724=1095.635,221.195,-72.510,177.291,18.192,152.428
C08725=1095.641,221.444,-72.535,177.295,18.193,152.428
C08726=1095.646,221.692,-72.559,177.297,18.194,152.428
C08727=1095.652,221.941,-72.585,177.301,18.196,152.427
C08728=1095.661,222.319,-72.623,177.306,18.198,152.427
C08729=1095.668,222.696,-72.661,177.310,18.200,152.426
C08730=1095.677,223.074,-72.700,177.315,18.201,152.426
C08731=1095.686,223.451,-72.738,177.319,18.203,152.426
C08732=1095.691,223.700,-72.764,177.323,18.205,152.425
C08733=1095.697,223.948,-72.788,177.326,18.206,152.425
C08734=1095.702,224.198,-72.814,177.330,18.208,152.425
C08735=1095.708,224.446,-72.839,177.332,18.209,152.424
C08736=1095.713,224.695,-72.865,177.336,18.211,152.424
C08737=1095.719,224.944,-72.890,177.339,18.212,152.424
C08738=1095.725,225.191,-72.915,177.342,18.213,152.423
C08739=1095.730,225.441,-72.940,177.345,18.215,152.423
C08740=1095.736,225.690,-72.965,177.349,18.216,152.423
C08741=1095.741,225.938,-72.991,177.351,18.217,152.423
C08742=1095.747,226.187,-73.016,177.355,18.219,152.422
C08743=1095.753,226.436,-73.042,177.358,18.220,152.422
C08744=1095.758,226.684,-73.067,177.361,18.222,152.422
C08745=1095.764,226.933,-73.093,177.364,18.223,152.421
C08746=1095.770,227.181,-73.119,177.368,18.224,152.421
C08747=1095.775,227.430,-73.143,177.371,18.225,152.421
C08748=1095.781,227.679,-73.169,177.373,18.227,152.421
C08749=1095.786,227.928,-73.195,177.377,18.228,152.420
C08750=1095.792,228.177,-73.220,177.380,18.229,152.420
C08751=1095.797,228.425,-73.246,177.383,18.231,152.420
C08752=1095.804,228.673,-73.271,177.386,18.232,152.419
C08753=1095.809,228.922,-73.297,177.390,18.234,152.419
C08754=1095.815,229.170,-73.322,177.393,18.235,152.419
C08755=1095.820,229.419,-73.348,177.396,18.236,152.418
C08756=1095.826,229.668,-73.374,177.399,18.237,152.418
C08757=1095.832,229.917,-73.399,177.403,18.239,152.418
C08758=1095.838,230.165,-73.426,177.406,18.240,152.417
C08759=1095.843,230.413,-73.451,177.409,18.242,152.417
C08760=1095.849,230.662,-73.477,177.412,18.243,152.417
C08761=1095.854,230.911,-73.503,177.416,18.244,152.417
C08762=1095.860,231.160,-73.528,177.418,18.246,152.416
C08763=1095.865,231.408,-73.553,177.422,18.247,152.416
C08764=1095.871,231.657,-73.579,177.425,18.249,152.416
C08765=1095.877,231.906,-73.605,177.428,18.250,152.415
C08766=1095.882,232.155,-73.631,177.431,18.251,152.415
C08767=1095.887,232.403,-73.657,177.435,18.253,152.415
C08768=1095.894,232.651,-73.682,177.438,18.254,152.415
C08769=1095.899,232.900,-73.708,177.441,18.256,152.414
C08770=1095.905,233.149,-73.734,177.444,18.257,152.414
C08771=1095.910,233.398,-73.760,177.447,18.259,152.414
C08772=1095.916,233.646,-73.786,177.450,18.260,152.413
C08773=1095.921,233.895,-73.812,177.454,18.261,152.413
C08774=1095.927,234.143,-73.838,177.457,18.263,152.413
C08775=1095.933,234.392,-73.864,177.460,18.264,152.413
C08776=1095.938,234.641,-73.890,177.464,18.266,152.412
C08777=1095.944,234.889,-73.915,177.467,18.267,152.412
C08778=1095.949,235.138,-73.941,177.470,18.269,152.412
C08779=1095.955,235.386,-73.968,177.473,18.270,152.412
C08780=1095.964,235.756,-74.006,177.477,18.272,152.411
C08781=1095.972,236.125,-74.045,177.483,18.274,152.411
C08782=1095.980,236.493,-74.084,177.487,18.276,152.410
C08783=1095.988,236.862,-74.123,177.492,18.278,152.410
C08784=1095.994,237.111,-74.148,177.496,18.280,152.410
C08785=1096.000,237.360,-74.174,177.498,18.281,152.409
C08786=1096.005,237.608,-74.201,177.502,18.283,152.409
C08787=1096.011,237.857,-74.227,177.505,18.284,152.409
C08788=1096.017,238.105,-74.253,177.508,18.286,152.408
C08789=1096.022,238.354,-74.279,177.511,18.287,152.408
C08790=1096.027,238.602,-74.306,177.515,18.289,152.408
C08791=1096.033,238.851,-74.332,177.518,18.290,152.408
C08792=1096.038,239.099,-74.358,177.521,18.291,152.407
C08793=1096.044,239.348,-74.384,177.525,18.293,152.407
C08794=1096.050,239.597,-74.411,177.527,18.294,152.407
C08795=1096.056,239.845,-74.436,177.531,18.296,152.406
C08796=1096.062,240.094,-74.463,177.534,18.297,152.406
C08797=1096.067,240.342,-74.489,177.537,18.299,152.406
C08798=1096.073,240.591,-74.515,177.541,18.301,152.406
C08799=1096.079,240.839,-74.542,177.544,18.301,152.405
C08800=1096.084,241.088,-74.568,177.547,18.303,152.405
C08801=1096.090,241.337,-74.595,177.550,18.304,152.405
C08802=1096.096,241.585,-74.621,177.554,18.306,152.405
C08803=1096.101,241.834,-74.647,177.557,18.307,152.404
C08804=1096.107,242.082,-74.674,177.560,18.309,152.404
C08805=1096.113,242.331,-74.700,177.563,18.310,152.404
C08806=1096.118,242.580,-74.726,177.566,18.312,152.404
C08807=1096.124,242.828,-74.753,177.570,18.313,152.403
C08808=1096.129,243.077,-74.780,177.573,18.315,152.403
C08809=1096.135,243.325,-74.807,177.576,18.316,152.403
C08810=1096.140,243.574,-74.833,177.579,18.318,152.402
C08811=1096.146,243.823,-74.859,177.583,18.319,152.402
C08812=1096.152,244.071,-74.886,177.586,18.321,152.402
C08813=1096.158,244.319,-74.913,177.589,18.322,152.402
C08814=1096.163,244.568,-74.939,177.593,18.324,152.401
C08815=1096.168,244.817,-74.966,177.595,18.325,152.401
C08816=1096.174,245.065,-74.993,177.599,18.327,152.401
C08817=1096.180,245.314,-75.019,177.602,18.329,152.401
C08818=1096.185,245.562,-75.046,177.605,18.330,152.400
C08819=1096.191,245.810,-75.073,177.609,18.332,152.400
C08820=1096.196,246.059,-75.100,177.611,18.333,152.400
C08821=1096.202,246.307,-75.126,177.615,18.334,152.399
C08822=1096.207,246.556,-75.152,177.619,18.336,152.399
C08823=1096.213,246.805,-75.179,177.621,18.337,152.399
C08824=1096.218,247.053,-75.206,177.625,18.339,152.399
C08825=1096.224,247.302,-75.233,177.627,18.341,152.398
C08826=1096.230,247.550,-75.260,177.631,18.342,152.398
C08827=1096.235,247.799,-75.287,177.635,18.344,152.398
C08828=1096.241,248.047,-75.313,177.637,18.345,152.398
C08829=1096.246,248.295,-75.340,177.641,18.347,152.397
C08830=1096.251,248.544,-75.367,177.645,18.349,152.397
C08831=1096.257,248.793,-75.394,177.647,18.350,152.397
C08832=1096.266,249.194,-75.437,177.652,18.353,152.397
C08833=1096.275,249.595,-75.481,177.658,18.355,152.396
C08834=1096.284,249.996,-75.525,177.663,18.358,152.396
C08835=1096.293,250.397,-75.569,177.668,18.361,152.395
C08836=1096.299,250.646,-75.595,177.671,18.362,152.395
C08837=1096.304,250.894,-75.623,177.675,18.364,152.395
C08838=1096.310,251.143,-75.649,177.677,18.365,152.395
C08839=1096.315,251.391,-75.677,177.681,18.367,152.394
C08840=1096.321,251.639,-75.704,177.685,18.368,152.394
C08841=1096.326,251.888,-75.731,177.687,18.369,152.394
C08842=1096.332,252.137,-75.758,177.691,18.371,152.394
C08843=1096.338,252.385,-75.785,177.694,18.373,152.393
C08844=1096.343,252.633,-75.813,177.697,18.374,152.393
C08845=1096.349,252.882,-75.839,177.701,18.376,152.393
C08846=1096.354,253.130,-75.867,177.704,18.378,152.393
C08847=1096.360,253.379,-75.893,177.707,18.379,152.392
C08848=1096.365,253.608,-75.919,177.710,18.381,152.392
C08849=1096.371,253.837,-75.944,177.713,18.382,152.392
C08850=1096.375,254.066,-75.969,177.716,18.384,152.392
C08851=1096.381,254.294,-75.994,177.719,18.385,152.391
C08852=1096.386,254.524,-76.019,177.722,18.387,152.391
C08853=1096.391,254.753,-76.045,177.726,18.388,152.391
C08854=1096.396,254.981,-76.070,177.728,18.390,152.391
C08855=1096.402,255.211,-76.096,177.731,18.391,152.391
C08856=1096.407,255.459,-76.122,177.734,18.393,152.390
C08857=1096.412,255.708,-76.149,177.738,18.395,152.390
C08858=1096.419,255.955,-76.177,177.741,18.396,152.390
C08859=1096.424,256.204,-76.204,177.744,18.398,152.390
C08860=1096.430,256.453,-76.232,177.748,18.399,152.389
C08861=1096.435,256.701,-76.259,177.750,18.401,152.389
C08862=1096.441,256.949,-76.287,177.754,18.403,152.389
C08863=1096.447,257.198,-76.314,177.757,18.404,152.389
C08864=1096.452,257.446,-76.342,177.760,18.406,152.388
C08865=1096.458,257.695,-76.369,177.764,18.407,152.388
C08866=1096.463,257.943,-76.397,177.767,18.409,152.388
C08867=1096.469,258.192,-76.424,177.770,18.411,152.388
C08868=1096.475,258.440,-76.451,177.773,18.412,152.387
C08869=1096.480,258.689,-76.479,177.777,18.414,152.387
C08870=1096.487,258.937,-76.506,177.780,18.415,152.387
C08871=1096.492,259.186,-76.534,177.783,18.417,152.387
C08872=1096.497,259.434,-76.562,177.787,18.419,152.387
C08873=1096.504,259.682,-76.589,177.789,18.420,152.386
C08874=1096.509,259.931,-76.617,177.793,18.422,152.386
C08875=1096.514,260.179,-76.645,177.796,18.424,152.386
C08876=1096.521,260.427,-76.672,177.799,18.425,152.385
C08877=1096.526,260.676,-76.700,177.803,18.427,152.385
C08878=1096.532,260.925,-76.728,177.806,18.428,152.385
C08879=1096.538,261.173,-76.755,177.810,18.430,152.385
C08880=1096.543,261.421,-76.783,177.813,18.431,152.385
C08881=1096.549,261.670,-76.811,177.816,18.433,152.384
C08882=1096.555,261.918,-76.838,177.820,18.435,152.384
C08883=1096.561,262.166,-76.867,177.822,18.436,152.384
C08884=1096.569,262.526,-76.906,177.828,18.439,152.384
C08885=1096.577,262.885,-76.946,177.832,18.441,152.383
C08886=1096.585,263.245,-76.987,177.837,18.444,152.383
C08887=1096.594,263.603,-77.027,177.842,18.446,152.382
C08888=1096.600,263.852,-77.055,177.845,18.447,152.382
C08889=1096.606,264.100,-77.082,177.848,18.449,152.382
C08890=1096.611,264.348,-77.110,177.852,18.451,152.382
C08891=1096.617,264.597,-77.139,177.855,18.453,152.381
C08892=1096.622,264.845,-77.167,177.858,18.454,152.381
C08893=1096.628,265.094,-77.195,177.861,18.456,152.381
C08894=1096.633,265.342,-77.222,177.865,18.458,152.381
C08895=1096.639,265.591,-77.251,177.868,18.460,152.381
C08896=1096.645,265.839,-77.279,177.871,18.461,152.380
C08897=1096.651,266.087,-77.306,177.874,18.463,152.380
C08898=1096.657,266.335,-77.334,177.878,18.465,152.380
C08899=1096.662,266.584,-77.362,177.881,18.466,152.380
C08900=1096.668,266.832,-77.391,177.884,18.468,152.380
C08901=1096.673,267.080,-77.419,177.887,18.470,152.379
C08902=1096.679,267.329,-77.447,177.891,18.472,152.379
C08903=1096.684,267.577,-77.475,177.894,18.473,152.379
C08904=1096.690,267.826,-77.503,177.897,18.475,152.379
C08905=1096.696,268.074,-77.531,177.901,18.477,152.379
C08906=1096.702,268.322,-77.560,177.904,18.479,152.378
C08907=1096.707,268.570,-77.588,177.907,18.480,152.378
C08908=1096.713,268.818,-77.616,177.910,18.482,152.378
C08909=1096.719,269.067,-77.644,177.914,18.484,152.378
C08910=1096.725,269.316,-77.673,177.917,18.486,152.377
C08911=1096.730,269.564,-77.701,177.920,18.487,152.377
C08912=1096.735,269.813,-77.730,177.924,18.489,152.377
C08913=1096.741,270.060,-77.758,177.927,18.491,152.377
C08914=1096.747,270.309,-77.787,177.930,18.493,152.377
C08915=1096.752,270.557,-77.815,177.933,18.495,152.377
C08916=1096.758,270.806,-77.843,177.937,18.496,152.376
C08917=1096.763,271.054,-77.871,177.940,18.498,152.376
C08918=1096.770,271.302,-77.900,177.944,18.500,152.376
C08919=1096.775,271.550,-77.928,177.947,18.502,152.376
C08920=1096.781,271.799,-77.956,177.950,18.504,152.375
C08921=1096.786,272.046,-77.985,177.953,18.505,152.375
C08922=1096.792,272.295,-78.014,177.957,18.507,152.375
C08923=1096.797,272.543,-78.042,177.960,18.509,152.375
C08924=1096.803,272.792,-78.070,177.963,18.511,152.375
C08925=1096.809,273.040,-78.099,177.966,18.513,152.374
C08926=1096.814,273.289,-78.128,177.970,18.514,152.374
C08927=1096.820,273.537,-78.157,177.973,18.517,152.374
C08928=1096.825,273.785,-78.185,177.976,18.519,152.374
C08929=1096.831,274.033,-78.213,177.979,18.520,152.374
C08930=1096.838,274.282,-78.242,177.983,18.522,152.373
C08931=1096.842,274.530,-78.271,177.986,18.524,152.373
C08932=1096.848,274.778,-78.300,177.989,18.526,152.373
C08933=1096.854,275.026,-78.328,177.992,18.527,152.373
C08934=1096.859,275.275,-78.357,177.995,18.529,152.373
C08935=1096.865,275.523,-78.385,177.999,18.531,152.373
C08936=1096.873,275.885,-78.427,178.004,18.534,152.372
C08937=1096.881,276.246,-78.469,178.008,18.536,152.372
C08938=1096.890,276.609,-78.511,178.013,18.539,152.372
C08939=1096.898,276.970,-78.553,178.018,18.542,152.372
C08940=1096.904,277.219,-78.582,178.021,18.544,152.371
C08941=1096.910,277.467,-78.611,178.025,18.546,152.371
C08942=1096.914,277.716,-78.639,178.028,18.548,152.371
C08943=1096.921,277.964,-78.668,178.032,18.550,152.371
C08944=1096.926,278.211,-78.697,178.034,18.551,152.371
C08945=1096.931,278.460,-78.726,178.038,18.553,152.371
C08946=1096.938,278.709,-78.755,178.041,18.555,152.370
C08947=1096.943,278.957,-78.785,178.044,18.557,152.370
C08948=1096.949,279.205,-78.813,178.048,18.559,152.370
C08949=1096.955,279.453,-78.842,178.050,18.561,152.370
C08950=1096.960,279.702,-78.871,178.054,18.563,152.370
C08951=1096.966,279.949,-78.900,178.057,18.564,152.369
C08952=1096.971,280.198,-78.929,178.061,18.567,152.369
C08953=1096.977,280.446,-78.958,178.064,18.569,152.369
C08954=1096.983,280.695,-78.988,178.067,18.571,152.369
C08955=1096.989,280.942,-79.016,178.070,18.572,152.369
C08956=1096.994,281.191,-79.045,178.074,18.574,152.369
C08957=1097.000,281.439,-79.074,178.077,18.576,152.369
C08958=1097.005,281.687,-79.103,178.080,18.578,152.368
C08959=1097.011,281.935,-79.133,178.084,18.580,152.368
C08960=1097.017,282.184,-79.162,178.087,18.582,152.368
C08961=1097.022,282.432,-79.192,178.090,18.584,152.368
C08962=1097.028,282.680,-79.220,178.093,18.586,152.368
C08963=1097.033,282.929,-79.249,178.096,18.588,152.368
C08964=1097.039,283.177,-79.278,178.100,18.590,152.367
C08965=1097.045,283.425,-79.308,178.103,18.592,152.367
C08966=1097.050,283.673,-79.337,178.106,18.594,152.367
C08967=1097.056,283.921,-79.366,178.110,18.596,152.367
C08968=1097.062,284.169,-79.396,178.112,18.598,152.367
C08969=1097.067,284.418,-79.426,178.116,18.600,152.367
C08970=1097.073,284.665,-79.454,178.119,18.602,152.367
C08971=1097.078,284.914,-79.484,178.123,18.604,152.366
C08972=1097.084,285.162,-79.514,178.126,18.606,152.366
C08973=1097.090,285.410,-79.543,178.130,18.608,152.366
C08974=1097.095,285.659,-79.572,178.133,18.610,152.366
C08975=1097.100,285.907,-79.602,178.136,18.612,152.366
C08976=1097.107,286.155,-79.631,178.139,18.614,152.366
C08977=1097.112,286.403,-79.660,178.142,18.616,152.365
C08978=1097.118,286.652,-79.690,178.146,18.618,152.365
C08979=1097.124,286.899,-79.720,178.149,18.620,152.365
C08980=1097.130,287.147,-79.749,178.152,18.622,152.365
C08981=1097.135,287.395,-79.778,178.156,18.624,152.365
C08982=1097.140,287.644,-79.808,178.159,18.626,152.365
C08983=1097.146,287.892,-79.837,178.162,18.628,152.365
C08984=1097.152,288.140,-79.867,178.165,18.630,152.365
C08985=1097.158,288.388,-79.897,178.168,18.632,152.364
C08986=1097.164,288.636,-79.926,178.172,18.634,152.364
C08987=1097.169,288.885,-79.956,178.175,18.636,152.364
C08988=1097.177,289.255,-80.001,178.180,18.639,152.364
C08989=1097.186,289.627,-80.045,178.185,18.642,152.364
C08990=1097.195,289.999,-80.089,178.190,18.646,152.364
C08991=1097.203,290.369,-80.134,178.194,18.648,152.363
C08992=1097.208,290.618,-80.163,178.198,18.650,152.363
C08993=1097.214,290.866,-80.193,178.201,18.652,152.363
C08994=1097.220,291.114,-80.223,178.204,18.655,152.363
C08995=1097.226,291.362,-80.253,178.208,18.657,152.363
C08996=1097.232,291.610,-80.283,178.211,18.659,152.363
C08997=1097.237,291.858,-80.312,178.214,18.661,152.363
C08998=1097.243,292.107,-80.342,178.218,18.663,152.363
C08999=1097.249,292.355,-80.372,178.221,18.666,152.363
C09000=1097.254,292.603,-80.402,178.224,18.668,152.362
C09001=1097.260,292.851,-80.432,178.228,18.670,152.362
C09002=1097.265,293.099,-80.462,178.231,18.672,152.362
C09003=1097.271,293.347,-80.492,178.234,18.674,152.362
C09004=1097.277,293.596,-80.522,178.237,18.676,152.362
C09005=1097.283,293.843,-80.552,178.240,18.678,152.362
C09006=1097.288,294.092,-80.582,178.244,18.680,152.362
C09007=1097.294,294.340,-80.612,178.247,18.682,152.362
C09008=1097.299,294.588,-80.642,178.250,18.685,152.362
C09009=1097.305,294.835,-80.672,178.253,18.687,152.361
C09010=1097.311,295.084,-80.703,178.257,18.689,152.361
C09011=1097.317,295.332,-80.732,178.260,18.691,152.361
C09012=1097.322,295.580,-80.763,178.263,18.693,152.361
C09013=1097.328,295.829,-80.792,178.267,18.696,152.361
C09014=1097.334,296.076,-80.823,178.270,18.698,152.361
C09015=1097.340,296.324,-80.853,178.273,18.700,152.361
C09016=1097.345,296.573,-80.883,178.277,18.702,152.361
C09017=1097.351,296.820,-80.913,178.280,18.704,152.361
C09018=1097.357,297.068,-80.943,178.283,18.707,152.361
C09019=1097.361,297.317,-80.974,178.286,18.709,152.360
C09020=1097.367,297.565,-81.004,178.290,18.711,152.360
C09021=1097.373,297.813,-81.034,178.293,18.713,152.360
C09022=1097.379,298.060,-81.065,178.296,18.716,152.360
C09023=1097.384,298.309,-81.094,178.300,18.718,152.360
C09024=1097.390,298.557,-81.125,178.303,18.720,152.360
C09025=1097.395,298.805,-81.156,178.306,18.722,152.360
C09026=1097.401,299.053,-81.186,178.309,18.725,152.360
C09027=1097.407,299.301,-81.216,178.313,18.727,152.360
C09028=1097.412,299.549,-81.247,178.316,18.729,152.360
C09029=1097.418,299.797,-81.277,178.319,18.732,152.360
C09030=1097.423,300.045,-81.307,178.322,18.734,152.360
C09031=1097.428,300.293,-81.338,178.326,18.736,152.360
C09032=1097.434,300.541,-81.369,178.329,18.738,152.360
C09033=1097.440,300.789,-81.399,178.332,18.741,152.359
C09034=1097.445,301.037,-81.430,178.335,18.743,152.359
C09035=1097.451,301.285,-81.460,178.338,18.746,152.359
C09036=1097.456,301.533,-81.491,178.342,18.748,152.359
C09037=1097.462,301.781,-81.522,178.345,18.750,152.359
C09038=1097.468,302.029,-81.552,178.348,18.753,152.359
C09039=1097.473,302.277,-81.583,178.351,18.755,152.359
C09040=1097.483,302.662,-81.631,178.356,18.758,152.359
C09041=1097.490,303.047,-81.678,178.361,18.762,152.359
C09042=1097.500,303.432,-81.725,178.366,18.766,152.359
C09043=1097.508,303.818,-81.773,178.372,18.770,152.359
C09044=1097.514,304.066,-81.804,178.375,18.772,152.359
C09045=1097.519,304.314,-81.835,178.378,18.774,152.359
C09046=1097.525,304.562,-81.865,178.381,18.776,152.359
C09047=1097.531,304.810,-81.897,178.384,18.779,152.359
C09048=1097.536,305.058,-81.927,178.388,18.781,152.359
C09049=1097.542,305.306,-81.958,178.391,18.784,152.359
C09050=1097.547,305.554,-81.989,178.394,18.786,152.359
C09051=1097.554,305.802,-82.019,178.397,18.788,152.359
C09052=1097.559,306.050,-82.051,178.401,18.791,152.359
C09053=1097.565,306.297,-82.081,178.404,18.793,152.359
C09054=1097.570,306.546,-82.112,178.407,18.795,152.358
C09055=1097.576,306.793,-82.143,178.410,18.798,152.358
C09056=1097.582,307.042,-82.175,178.414,18.800,152.358
C09057=1097.588,307.289,-82.205,178.417,18.803,152.358
C09058=1097.593,307.538,-82.236,178.420,18.805,152.358
C09059=1097.599,307.785,-82.266,178.423,18.807,152.358
C09060=1097.605,308.034,-82.298,178.426,18.810,152.358
C09061=1097.610,308.281,-82.329,178.430,18.813,152.358
C09062=1097.616,308.529,-82.360,178.433,18.815,152.358
C09063=1097.621,308.778,-82.392,178.437,18.817,152.358
C09064=1097.627,309.026,-82.422,178.440,18.820,152.358
C09065=1097.633,309.273,-82.454,178.443,18.822,152.358
C09066=1097.639,309.522,-82.484,178.446,18.825,152.358
C09067=1097.644,309.769,-82.516,178.450,18.827,152.358
C09068=1097.650,310.017,-82.546,178.453,18.830,152.358
C09069=1097.656,310.265,-82.579,178.456,18.832,152.358
C09070=1097.661,310.513,-82.609,178.459,18.834,152.358
C09071=1097.667,310.761,-82.640,178.462,18.837,152.358
C09072=1097.673,311.009,-82.672,178.465,18.839,152.358
C09073=1097.679,311.257,-82.703,178.469,18.842,152.358
C09074=1097.684,311.505,-82.734,178.472,18.844,152.358
C09075=1097.690,311.753,-82.766,178.476,18.847,152.358
C09076=1097.696,312.001,-82.796,178.479,18.849,152.358
C09077=1097.702,312.249,-82.828,178.482,18.852,152.358
C09078=1097.707,312.497,-82.859,178.485,18.854,152.358
C09079=1097.713,312.744,-82.890,178.489,18.857,152.358
C09080=1097.719,312.993,-82.922,178.492,18.859,152.358
C09081=1097.724,313.241,-82.953,178.495,18.862,152.358
C09082=1097.731,313.489,-82.985,178.498,18.864,152.358
C09083=1097.737,313.736,-83.016,178.501,18.867,152.358
C09084=1097.742,313.985,-83.048,178.504,18.869,152.358
C09085=1097.748,314.232,-83.079,178.507,18.872,152.358
C09086=1097.754,314.480,-83.111,178.511,18.875,152.358
C09087=1097.759,314.728,-83.142,178.515,18.877,152.358
C09088=1097.766,314.976,-83.173,178.518,18.880,152.358
C09089=1097.771,315.224,-83.205,178.521,18.882,152.358
C09090=1097.777,315.472,-83.237,178.524,18.885,152.358
C09091=1097.783,315.720,-83.268,178.527,18.887,152.358
C09092=1097.791,316.108,-83.318,178.532,18.892,152.358
C09093=1097.800,316.496,-83.367,178.537,18.896,152.358
C09094=1097.808,316.883,-83.417,178.542,18.899,152.358
